(*------------------------------------------------------------------------------------------Modbus TCP Functions---------------------------------------------------------------------------------------------*)

fbMBRead_FC3(	sIPAddr:= str_IPAdress, 
				nTCPPort:= 502,
				cbLength:= SIZEOF(arrBuffer_FC3), 
				pDestAddr:= ADR(arrBuffer_FC3), 
				tTimeout:= T#10S,
				nErrId => udint_Error_ID);

FPError_FC_3(CLK:= fbMBRead_FC3.  bError, Q=> );		

(*------------------------------------------------------------------------------------------State Machine Error---------------------------------------------------------------------------------------------*)	

CASE iStateModbusError OF
	
	300://Error
		timer_Wait.IN :=TRUE;
		timer_Delay.IN := FALSE;
		fbMBRead_FC3.bExecute := FALSE;
		m_MBTCPError := TRUE; 		
		m_Poll_ok:=FALSE;
		int_Data_Received:=0;
				//Restart from new with the Read out part after an Error
		IF timer_Wait.Q = TRUE THEN
			iStateModbusRead := 0;	
			iStateModbusError := 0;
			timer_Wait.IN :=FALSE;
			timer_Timeout.IN := FALSE;
		END_IF		
							
END_CASE

END_FUNCTION_BLOCK

// ---- FBs/General/FB_ModBus_2Registers_FC4.TcPOU
FUNCTION_BLOCK FB_ModBus_2Registers_FC4
VAR_INPUT PERSISTENT
	m_Enable					: BOOL;						//Enable the Fuctionblock and his logic
	str_IPAdress				: STRING(15);				//IP Adress of the meter
	w_Adress					: WORD;						//modbus adress
	int_Divider					: INT;						//Devider of the received data
	n_UnitID					: BYTE:=255;				// dentification number of a serial sub-network device. If a device is addressed directly via TCP/IP, this value must be 16#FF / 255
	m_Float32Conversion			: BOOL;						// receives value in Float 32 / real format
	m_LittleEndian				: BOOL;

END_VAR
VAR_OUTPUT
	m_PollSuccessful			: BOOL;						//Poll succesfull		
	r_ReceivedValue				: REAL;						//Received Value
	udint_Error_ID				: UDINT;					// ERR ID FB_MBReadRegs
END_VAR
VAR
	{attribute 'hide'}
	timer_Delay					: TON;						//Timer for Delay between Requests
	{attribute 'hide'}
	timer_DelayStart			: TON;						//Timer to start the state machine with Delay after enabling or after the system ist restartet
	{attribute 'hide'}
	timer_TimeOut				: TON;						//Timer for Timeout MB Read
	{attribute 'hide'}
	iStateModbusRead			: INT;						//State machine for read out Data over Modbus RTU
	{attribute 'hide'}
	fbMBRead_FC4				: FB_MBReadInputRegs  ;		//Modbus Read Function (FC4)
	{attribute 'hide'}
	ftrig_PEnable				: f_trig;					//Internal positive Edge
	{attribute 'hide'}
	iStateModbusError			: INT;						//State machine for error out Data over Modbus TCP/IP	
	{attribute 'hide'}
	FPError_FC4				: R_TRIG;					//Internal positive Edge
	{attribute 'hide'}
	arrBuffer_FC4				: ARRAY[1..2] OF WORD;		//Buffer with Data from FC4
	{attribute 'hide'}
	timer_Connection_ok			: TON;
	int_Data_Received			: INT;
	{attribute 'hide'}
	m_MBTCPError				: BOOL;
	{attribute 'hide'}
	int_Data_Received_old		: INT;
	{attribute 'hide'}
	timer_Connection_ok_TOF	: TOF;
	{attribute 'hide'}
	fbConvertWordToDword		: FB_CV_WORD_TO_DWORD;			//Convert Word to Dword
	{attribute 'hide'}
	usintSign					: USINT;						// converstion dword to real	
	{attribute 'hide'}
	intExponent					: INT;							// converstion dword to real
	{attribute 'hide'}
	realMantisse				: REAL;							// converstion dword to real
	{attribute 'hide'}
	m_Poll_ok: BOOL;
	{attribute 'hide'}
	timer_Wait: Ton;
	int_TimeoutError: INT;
	int_FC4Error: INT;
END_VAR

(*--------------------------------------------------------------------------------------------Limits-------------------------------------------------------------------------------------*)

w_Adress := LIMIT(0,w_Adress,65535);
int_Divider := LIMIT(1,int_Divider,32767);
	
(*--------------------------------------------------------------------------------------------State Machine Read--------------------------------------------------------------------------------------*)

//Timer for Delay
timer_Delay(IN:= , PT:= T#50MS, Q=> , ET=> );

//Timeout Timer is dissabled when the Init Step is aktiv or the function is not enabled
IF iStateModbusRead = 0 OR NOT m_Enable THEN 
	timer_Timeout.IN := FALSE; 
END_IF
timer_Timeout(IN:= , PT:= T#1S, Q=> , ET=> );

//Enable with Delay that not all sockets have to be created at the same time
timer_DelayStart(IN:= m_Enable, PT:= T#1S, Q=> , ET=> );
ftrig_PEnable(CLK:= timer_DelayStart.Q, Q=> );

IF ftrig_PEnable.Q AND iStateModbusRead = 0 THEN 
	iStateModbusRead := 1; 
END_IF		
		
//Not Enabled
IF NOT m_Enable THEN 
	iStateModbusRead := 0; 
	iStateModbusError := 0; 
END_IF		
		
CASE iStateModbusRead OF

	0://Init Step 
		timer_Delay.IN := FALSE;
		fbMBRead_FC4.bExecute := FALSE;
		m_Poll_ok:=FALSE;
		int_Data_Received:=0;
	
		iStateModbusRead := 1;
	
	1://read the required registers
		//Start Read
		fbMBRead_FC4.nQuantity := 2;
		fbMBRead_FC4.nMBAddr := w_Adress;
		fbMBRead_FC4.bExecute := TRUE;
		fbMBRead_FC4.nUnitID := n_UnitID;
		timer_Timeout.IN := TRUE;
		IF fbMBRead_FC4.bBusy THEN 
			timer_Delay.IN := TRUE; 
		END_IF
		
		//Wait for Delay, copy Data and then next step
		IF NOT fbMBRead_FC4.bBusy AND NOT fbMBRead_FC4.bError AND timer_Delay.Q THEN
			m_Poll_ok:=TRUE;
			int_Data_Received:=int_Data_Received+1;
			m_MBTCPError := FALSE; 
			// convert received data
			IF m_Float32Conversion AND NOT m_LittleEndian THEN
		//		fbConvertWordToDword(wInputValue_1:= arrBuffer_FC4[1], wInputValue_2:= arrBuffer_FC4[2], eByteOrderForConvert:= eByteOrder.eLittleEndian , dwOutputValue=> );
				fbConvertWordToDword(wInputValue_1:= arrBuffer_FC4[1], wInputValue_2:= arrBuffer_FC4[2], eByteOrderForConvert:= eByteOrder.eBigEndian , dwOutputValue=> );
				(* Sign *)
				usintSign:=BOOL_TO_USINT(fbConvertWordToDword.dwOutputValue.31);
				(* Exponent *)
				intExponent:=DWORD_TO_INT(SHR(fbConvertWordToDword.dwOutputValue,23) AND 16#FF);
				(* Mantisse *)
				realMantisse:=DWORD_TO_REAL(fbConvertWordToDword.dwOutputValue AND 16#7FFFFF);
				(* Result *)
				r_ReceivedValue := LREAL_TO_REAL((EXPT((-1),usintSign) * (1+realMantisse/8388608) * EXPT(2,intExponent-127))/int_Divider);
			ELSIF m_Float32Conversion AND m_LittleEndian THEN
				fbConvertWordToDword(wInputValue_1:= arrBuffer_FC4[1], wInputValue_2:= arrBuffer_FC4[2], eByteOrderForConvert:= eByteOrder.eLittleEndian , dwOutputValue=> );
				(* Sign *)
				usintSign:=BOOL_TO_USINT(fbConvertWordToDword.dwOutputValue.31);
				(* Exponent *)
				intExponent:=DWORD_TO_INT(SHR(fbConvertWordToDword.dwOutputValue,23) AND 16#FF);
				(* Mantisse *)
				realMantisse:=DWORD_TO_REAL(fbConvertWordToDword.dwOutputValue AND 16#7FFFFF);
				(* Result *)
				r_ReceivedValue := LREAL_TO_REAL((EXPT((-1),usintSign) * (1+realMantisse/8388608) * EXPT(2,intExponent-127))/int_Divider);
			ELSE
				fbConvertWordToDword(wInputValue_1:= arrBuffer_FC4[2], wInputValue_2:= arrBuffer_FC4[1], eByteOrderForConvert:= eByteOrder.eLittleEndian , dwOutputValue=> );
				r_ReceivedValue := DINT_TO_REAL(fbConvertWordToDword.dwOutputValue)/int_Divider;
			END_IF
			
			//Go to Next Step
			timer_Timeout.IN := FALSE;
			fbMBRead_FC4.bExecute := FALSE;
			timer_Delay.IN := FALSE;		
			iStateModbusRead := 3;
		END_IF	

		//Error or Timeout
		IF FPError_FC4.Q THEN 
			iStateModbusError := 300;
			int_FC4Error := int_FC4Error+1;
		ELSIF timer_Timeout.Q THEN 
			timer_Timeout.IN := FALSE; 	  	
			iStateModbusError := 300;
			int_TimeoutError := int_TimeoutError+1;
		END_IF
		
	
	3://Wait and go to step 1
		//1 because 0 is the Init Step for Read
		timer_Wait.IN := TRUE;
		
		IF timer_Wait.Q = TRUE THEN
			iStateModbusRead := 1;
			timer_Wait.IN :=FALSE;
		END_IF

			
		
		//Error on Master, changes on Inputs or Timeout
		IF timer_Timeout.Q THEN 
			iStateModbusError := 300; 
		END_IF
	
END_CASE

(* wait timer*)

timer_Wait(PT:=T#3S);


(*------------------------------------------------------------------Error and Warning----------------------------------------------------------------------------*)	
 
timer_Connection_ok			(In:=int_Data_Received<>int_Data_Received_old,PT:=T#10S);
timer_Connection_ok_TOF		(In:=NOT(int_Data_Received<>int_Data_Received_old) AND int_Data_Received>3 ,PT:=T#20S);
int_Data_Received_old:=int_Data_Received;
m_PollSuccessful:=NOT timer_Connection_ok.Q AND timer_Connection_ok_TOF.Q ;

(*------------------------------------------------------------------------------------------Modbus TCP Functions---------------------------------------------------------------------------------------------*)

fbMBRead_FC4(	sIPAddr:= str_IPAdress, 
				nTCPPort:= 502,
				cbLength:= SIZEOF(arrBuffer_FC4), 
				pDestAddr:= ADR(arrBuffer_FC4), 
				tTimeout:= T#10S,
				nErrId => udint_Error_ID);

FPError_FC4(CLK:= fbMBRead_FC4.  bError, Q=> );		

(*------------------------------------------------------------------------------------------State Machine Error---------------------------------------------------------------------------------------------*)	

CASE iStateModbusError OF
	
	300://Error
		timer_Wait.IN :=TRUE;
		timer_Delay.IN := FALSE;
		fbMBRead_FC4.bExecute := FALSE;
		m_MBTCPError := TRUE; 		
		m_Poll_ok:=FALSE;
		int_Data_Received:=0;
				//Restart from new with the Read out part after an Error
		IF timer_Wait.Q = TRUE THEN
			iStateModbusRead := 0;	
			iStateModbusError := 0;
			timer_Wait.IN :=FALSE;
			timer_Timeout.IN := FALSE;
		END_IF		
							
END_CASE

END_FUNCTION_BLOCK

// ---- FBs/GMC Instruments/FB_EM2289.TcPOU
FUNCTION_BLOCK FB_EM2289
VAR_INPUT PERSISTENT
	m_Enable					: BOOL;						//Enable the Fuctionblock and his logic
	str_IPAdress				: STRING(15);				//IP Adress of the meter
END_VAR
VAR_OUTPUT
	real_RealPower_kW				: REAL;					// Real power in W
	real_RealPowerL1_kW				: REAL;					// Real power in W
	real_RealPowerL2_kW				: REAL;					// Real power in W
	real_RealPowerL3_kW				: REAL;					// Real power in W
	real_ReactivePower_kVAr			: REAL;					// Reactive power in VAr
	real_ApparentPower_kVA			: REAL;					// Apparent power in VA
	real_Frequency_Hz				: REAL;					// Frequency in Hz
	real_VoltageL1N_V				: REAL;					//  Voltage L1-N in V 
	real_VoltageL2N_V				: REAL;					//  Voltage L2-N in V 
	real_VoltageL3N_V				: REAL;					//  Voltage L3-N in V 
	real_VoltageL1L2_V				: REAL;					//  Voltage L1-L2 in V 
	real_VoltageL2L3_V				: REAL;					//  Voltage L2-L3 in V 
	real_VoltageL3L1_V				: REAL;					//  Voltage L3-L1 in V 
	real_CurrentL1_A				: REAL;					//  Current L1 in A
	real_CurrentL2_A				: REAL;					//  Current L2 in A
	real_CurrentL3_A				: REAL;					//  Current L3 in A
	real_EnergyTotal_Import_Wh		: REAL;					// Energy total in Wh
	real_EnergyTotal_Export_Wh		: REAL;					// Energy total in Wh
	real_EnergyTotal_ExportT1_Wh	: REAL;					// Energy total in Wh
	real_EnergyTotal_ExportT2_Wh	: REAL;					// Energy total in Wh
	m_PollSuccessful				: BOOL;					// Poll succesfull		
	udint_Error_ID					: UDINT;				// ERR ID FB_MBReadRegs
END_VAR
VAR
	{attribute 'hide'}
	w_Adress					: WORD;						//modbus adress
	{attribute 'hide'}
	usint_Quantity				: USINT;					//Number of Words to get polled, max 100
	{attribute 'hide'}
	fbConvertWordToDword		: FB_CV_WORD_TO_DWORD;			//Convert Word to Dword
	{attribute 'hide'}
	usintSign					: USINT;						// converstion dword to real	
	{attribute 'hide'}
	intExponent					: INT;							// converstion dword to real
	{attribute 'hide'}
	realMantisse				: REAL;							// converstion dword to real
	{attribute 'hide'}
	timer_Delay					: TON;						//Timer for Delay between Requests
	{attribute 'hide'}
	timer_DelayStart			: TON;						//Timer to start the state machine with Delay after enabling or after the system ist restartet
	{attribute 'hide'}
	timer_TimeOut				: TON;						//Timer for Timeout MB Read
	{attribute 'hide'}
	iStateModbusRead			: INT;						//State machine for read out Data over Modbus RTU
	{attribute 'hide'}
	fbMBRead_FC4				: FB_MBReadInputRegs  ;		//Modbus Read Function (FC4)
	{attribute 'hide'}
	ftrig_PEnable				: f_trig;					//Internal positive Edge
	{attribute 'hide'}
	iStateModbusError			: INT;						//State machine for error out Data over Modbus TCP/IP	
	{attribute 'hide'}
	FPError_FC_4				: R_TRIG;					//Internal positive Edge
	{attribute 'hide'}
	arrBuffer_FC4				: ARRAY[0..100] OF WORD;		//Buffer with Data from FC4
	{attribute 'hide'}
	timer_Connection_ok			: TON;
	{attribute 'hide'}
	int_Data_Received			: INT;
	{attribute 'hide'}
	m_MBTCPError				: BOOL;
	{attribute 'hide'}
	int_Data_Received_old		: INT;
	{attribute 'hide'}
	timer_Connection_ok_TOF	: TOF;
	{attribute 'hide'}
	m_Poll_ok: BOOL;
	{attribute 'hide'}
	timer_Wait: Ton;
	{attribute 'hide'}
	int_TimeoutError: INT;
	{attribute 'hide'}
	int_FC4Error: INT;
	{attribute 'hide'}
	i: INT;
	{attribute 'hide'}
	x: INT;
	sint_Exponent: SINT;
	real_EnergyFactor: REAL;
	
END_VAR

// v0.1 by Stefan Lackner 20230327
// not tested 
// reads out GMC Instruments EM2289   


(*--------------------------------------------------------------------------------------------Limits-------------------------------------------------------------------------------------*)
w_Adress := LIMIT(0,w_Adress,65000);
usint_Quantity := LIMIT(1,usint_Quantity,100);
	
(*--------------------------------------------------------------------------------------------State Machine Read--------------------------------------------------------------------------------------*)

//Timer for Delay
timer_Delay(IN:= , PT:= T#50MS, Q=> , ET=> );

//Timeout Timer is dissabled when the Init Step is aktiv or the function is not enabled
IF iStateModbusRead = 0 OR NOT m_Enable THEN 
	timer_Timeout.IN := FALSE; 
END_IF
timer_Timeout(IN:= , PT:= T#1S, Q=> , ET=> );

//Enable with Delay that not all sockets have to be created at the same time
timer_DelayStart(IN:= m_Enable, PT:= T#1S, Q=> , ET=> );
ftrig_PEnable(CLK:= timer_DelayStart.Q, Q=> );

IF ftrig_PEnable.Q AND iStateModbusRead = 0 THEN 
	iStateModbusRead := 1; 
END_IF		
		
//Not Enabled
IF NOT m_Enable THEN 
	iStateModbusRead := 0; 
	iStateModbusError := 0; 
END_IF		
		
CASE iStateModbusRead OF

	0://Init Step 
		timer_Delay.IN := FALSE;
		fbMBRead_FC4.bExecute := FALSE;
		m_Poll_ok:=FALSE;
		int_Data_Received:=0;
		iStateModbusRead := iStateModbusRead+1;

	1: // clean the array  Poll 1
		FOR i:=0 TO 100 BY 1 DO
			arrBuffer_FC4[i] := 0;
		END_FOR
		w_Adress := 0;
		usint_Quantity := 13; 
		iStateModbusRead := iStateModbusRead+1;
		
	2://read the required registers
		//Start Read Poll 1
		fbMBRead_FC4.nQuantity := usint_Quantity;
		fbMBRead_FC4.nMBAddr := w_Adress;
		fbMBRead_FC4.bExecute := TRUE;
		fbMBRead_FC4.nUnitID := 1;
		timer_Timeout.IN := TRUE;
		IF fbMBRead_FC4.bBusy THEN 
			timer_Delay.IN := TRUE; 
		END_IF
		
		//Wait for Delay, copy Data and then next step
		IF NOT fbMBRead_FC4.bBusy AND NOT fbMBRead_FC4.bError AND timer_Delay.Q THEN
			m_Poll_ok:=TRUE;
			int_Data_Received:=int_Data_Received+1;
			m_MBTCPError := FALSE; 
			
			//Go to Next Step
			timer_Timeout.IN := FALSE;
			fbMBRead_FC4.bExecute := FALSE;
			timer_Delay.IN := FALSE;		
			iStateModbusRead := iStateModbusRead+1;
		END_IF	

		//Error or Timeout
		IF FPError_FC_4.Q THEN 
			iStateModbusError := 300;
			int_FC4Error := int_FC4Error+1;
		ELSIF timer_Timeout.Q THEN  
			timer_Timeout.IN := FALSE; 	
			iStateModbusError := 300;
			int_TimeoutError := int_TimeoutError+1;
		END_IF
		
	3: // convert data Poll 1
		sint_Exponent := WORD_TO_SINT (arrBuffer_FC4[12]);
		real_VoltageL1L2_V := LREAL_TO_REAL(WORD_TO_REAL(arrBuffer_FC4[0])* EXPT (10,sint_Exponent));
		real_VoltageL2L3_V := LREAL_TO_REAL(WORD_TO_REAL(arrBuffer_FC4[1])* EXPT (10,sint_Exponent));
		real_VoltageL3L1_V := LREAL_TO_REAL(WORD_TO_REAL(arrBuffer_FC4[2])* EXPT (10,sint_Exponent));
		real_VoltageL1N_V :=  LREAL_TO_REAL(WORD_TO_REAL(arrBuffer_FC4[4])* EXPT (10,sint_Exponent));
		real_VoltageL2N_V :=  LREAL_TO_REAL(WORD_TO_REAL(arrBuffer_FC4[5])* EXPT (10,sint_Exponent));
		real_VoltageL3N_V :=  LREAL_TO_REAL(WORD_TO_REAL(arrBuffer_FC4[6])* EXPT (10,sint_Exponent));
		real_Frequency_Hz := WORD_TO_REAL(arrBuffer_FC4[11])/100;
		// go to next step
		iStateModbusRead := iStateModbusRead+1;
	
	4://Wait and go to next step
		timer_Wait.IN := TRUE;
		
		IF timer_Wait.Q = TRUE THEN
			iStateModbusRead := iStateModbusRead+1;
			timer_Wait.IN :=FALSE;
		END_IF

	5: // clean the array  Poll 2
		FOR i:=0 TO 100 BY 1 DO
			arrBuffer_FC4[i] := 0;
		END_FOR
		w_Adress := 100;
		usint_Quantity := 9; 
		iStateModbusRead := iStateModbusRead+1;
		
	6://read the required registers
		//Start Read  Poll 2
		fbMBRead_FC4.nQuantity := usint_Quantity;
		fbMBRead_FC4.nMBAddr := w_Adress;
		fbMBRead_FC4.bExecute := TRUE;
		fbMBRead_FC4.nUnitID := 1;
		timer_Timeout.IN := TRUE;
		IF fbMBRead_FC4.bBusy THEN 
			timer_Delay.IN := TRUE; 
		END_IF
		
		//Wait for Delay, copy Data and then next step
		IF NOT fbMBRead_FC4.bBusy AND NOT fbMBRead_FC4.bError AND timer_Delay.Q THEN
			m_Poll_ok:=TRUE;
			int_Data_Received:=int_Data_Received+1;
			m_MBTCPError := FALSE; 
			
			//Go to Next Step
			timer_Timeout.IN := FALSE;
			fbMBRead_FC4.bExecute := FALSE;
			timer_Delay.IN := FALSE;		
			iStateModbusRead := iStateModbusRead+1;
		END_IF	

		//Error or Timeout
		IF FPError_FC_4.Q THEN 
			iStateModbusError := 300;
			int_FC4Error := int_FC4Error+1;
		ELSIF timer_Timeout.Q THEN  
			timer_Timeout.IN := FALSE; 	
			iStateModbusError := 300;
			int_TimeoutError := int_TimeoutError+1;
		END_IF
		
	7: // convert data Poll 2
		sint_Exponent := WORD_TO_SINT (arrBuffer_FC4[8]);
		real_CurrentL1_A := LREAL_TO_REAL(WORD_TO_REAL(arrBuffer_FC4[0])* EXPT (10,sint_Exponent));
		real_CurrentL2_A := LREAL_TO_REAL(WORD_TO_REAL(arrBuffer_FC4[1])* EXPT (10,sint_Exponent));
		real_CurrentL3_A := LREAL_TO_REAL(WORD_TO_REAL(arrBuffer_FC4[2])* EXPT (10,sint_Exponent));
		
		// go to next step
		iStateModbusRead := iStateModbusRead+1;
			
		//Error on Master, changes on Inputs or Timeout
		IF timer_Timeout.Q THEN 
			iStateModbusError := 300; 
		END_IF
		
	8://Wait and go to next step
		timer_Wait.IN := TRUE;
		
		IF timer_Wait.Q = TRUE THEN
			iStateModbusRead := iStateModbusRead+1;
			timer_Wait.IN :=FALSE;
		END_IF

	9: // clean the array  Poll 3
		FOR i:=0 TO 100 BY 1 DO
			arrBuffer_FC4[i] := 0;
		END_FOR
		w_Adress := 200;
		usint_Quantity := 13; 
		iStateModbusRead := iStateModbusRead+1;
		
	10://read the required registers
		//Start Read  Poll 3
		fbMBRead_FC4.nQuantity := usint_Quantity;
		fbMBRead_FC4.nMBAddr := w_Adress;
		fbMBRead_FC4.bExecute := TRUE;
		fbMBRead_FC4.nUnitID := 1;
		timer_Timeout.IN := TRUE;
		IF fbMBRead_FC4.bBusy THEN 
			timer_Delay.IN := TRUE; 
		END_IF
		
		//Wait for Delay, copy Data and then next step
		IF NOT fbMBRead_FC4.bBusy AND NOT fbMBRead_FC4.bError AND timer_Delay.Q THEN
			m_Poll_ok:=TRUE;
			int_Data_Received:=int_Data_Received+1;
			m_MBTCPError := FALSE; 
			
			//Go to Next Step
			timer_Timeout.IN := FALSE;
			fbMBRead_FC4.bExecute := FALSE;
			timer_Delay.IN := FALSE;		
			iStateModbusRead := iStateModbusRead+1;
		END_IF	

		//Error or Timeout
		IF FPError_FC_4.Q THEN 
			iStateModbusError := 300;
			int_FC4Error := int_FC4Error+1;
		ELSIF timer_Timeout.Q THEN  
			timer_Timeout.IN := FALSE; 	
			iStateModbusError := 300;
			int_TimeoutError := int_TimeoutError+1;
		END_IF
		
	11: // convert data Poll 3
		sint_Exponent := WORD_TO_SINT (arrBuffer_FC4[12]);
		real_RealPowerL1_kW := LREAL_TO_REAL(WORD_TO_REAL(arrBuffer_FC4[0])* EXPT (10,sint_Exponent)/1000);
		real_RealPowerL2_kW := LREAL_TO_REAL(WORD_TO_REAL(arrBuffer_FC4[1])* EXPT (10,sint_Exponent)/1000);
		real_RealPowerL3_kW := LREAL_TO_REAL(WORD_TO_REAL(arrBuffer_FC4[2])* EXPT (10,sint_Exponent)/1000);
		real_RealPower_kW := LREAL_TO_REAL(WORD_TO_REAL(arrBuffer_FC4[3])* EXPT (10,sint_Exponent)/1000);
		real_RealPowerL1_kW := LREAL_TO_REAL(WORD_TO_REAL(arrBuffer_FC4[0])* EXPT (10,sint_Exponent)/1000);
		real_ReactivePower_kVAr := LREAL_TO_REAL(WORD_TO_REAL(arrBuffer_FC4[7])* EXPT (10,sint_Exponent)/1000);
		
		IF (real_RealPower_kW*real_RealPower_kW + real_ReactivePower_kVAr*real_ReactivePower_kVAr) <>0 THEN 
			real_ApparentPower_kVA := SQRT(ABS(real_RealPower_kW*real_RealPower_kW + real_ReactivePower_kVAr*real_ReactivePower_kVAr));	
		ELSE
	 		real_ApparentPower_kVA :=0;
		END_IF
		
		
		// go to next step
		iStateModbusRead := iStateModbusRead+1;
			
		//Error on Master, changes on Inputs or Timeout
		IF timer_Timeout.Q THEN 
			iStateModbusError := 300; 
		END_IF
		
	12://Wait and go to next step
		timer_Wait.IN := TRUE;
		
		IF timer_Wait.Q = TRUE THEN
			iStateModbusRead := iStateModbusRead+1;
			timer_Wait.IN :=FALSE;
		END_IF

	13: // clean the array  Poll 4
		FOR i:=0 TO 100 BY 1 DO
			arrBuffer_FC4[i] := 0;
		END_FOR
		w_Adress := 300;
		usint_Quantity := 10; 
		iStateModbusRead := iStateModbusRead+1;
		
	14://read the required registers
		//Start Read  Poll 4
		fbMBRead_FC4.nQuantity := usint_Quantity;
		fbMBRead_FC4.nMBAddr := w_Adress;
		fbMBRead_FC4.bExecute := TRUE;
		fbMBRead_FC4.nUnitID := 1;
		timer_Timeout.IN := TRUE;
		IF fbMBRead_FC4.bBusy THEN 
			timer_Delay.IN := TRUE; 
		END_IF
		
		//Wait for Delay, copy Data and then next step
		IF NOT fbMBRead_FC4.bBusy AND NOT fbMBRead_FC4.bError AND timer_Delay.Q THEN
			m_Poll_ok:=TRUE;
			int_Data_Received:=int_Data_Received+1;
			m_MBTCPError := FALSE; 
			
			//Go to Next Step
			timer_Timeout.IN := FALSE;
			fbMBRead_FC4.bExecute := FALSE;
			timer_Delay.IN := FALSE;		
			iStateModbusRead := iStateModbusRead+1;
		END_IF	

		//Error or Timeout
		IF FPError_FC_4.Q THEN 
			iStateModbusError := 300;
			int_FC4Error := int_FC4Error+1;
		ELSIF timer_Timeout.Q THEN  
			timer_Timeout.IN := FALSE; 	
			iStateModbusError := 300;
			int_TimeoutError := int_TimeoutError+1;
		END_IF
		
	15: // convert data Poll 4
		// energy factor
		fbConvertWordToDword(wInputValue_1:= arrBuffer_FC4[8], wInputValue_2:= arrBuffer_FC4[9], eByteOrderForConvert:= eByteOrder.eBigEndian , dwOutputValue=> );
		real_EnergyFactor := DWORD_TO_REAL (fbConvertWordToDword.dwOutputValue);
				
		fbConvertWordToDword(wInputValue_1:= arrBuffer_FC4[0], wInputValue_2:= arrBuffer_FC4[1], eByteOrderForConvert:= eByteOrder.eBigEndian , dwOutputValue=> );
		real_EnergyTotal_Import_Wh := DWORD_TO_REAL(fbConvertWordToDword.dwOutputValue) * real_EnergyFactor;
		
		fbConvertWordToDword(wInputValue_1:= arrBuffer_FC4[2], wInputValue_2:= arrBuffer_FC4[3], eByteOrderForConvert:= eByteOrder.eBigEndian , dwOutputValue=> );
		real_EnergyTotal_Export_Wh := DWORD_TO_REAL(fbConvertWordToDword.dwOutputValue) * real_EnergyFactor;
	
		// go to next step
		iStateModbusRead := iStateModbusRead+1;
			
		//Error on Master, changes on Inputs or Timeout
		IF timer_Timeout.Q THEN 
			iStateModbusError := 300; 
		END_IF		

	16://Wait and go to next step
		timer_Wait.IN := TRUE;
		
		IF timer_Wait.Q = TRUE THEN
			iStateModbusRead := iStateModbusRead+1;
			timer_Wait.IN :=FALSE;
		END_IF

	17: // clean the array  Poll 5
		FOR i:=0 TO 100 BY 1 DO
			arrBuffer_FC4[i] := 0;
		END_FOR
		w_Adress := 600;
		usint_Quantity := 10; 
		iStateModbusRead := iStateModbusRead+1;
		
	18://read the required registers
		//Start Read  Poll 5
		fbMBRead_FC4.nQuantity := usint_Quantity;
		fbMBRead_FC4.nMBAddr := w_Adress;
		fbMBRead_FC4.bExecute := TRUE;
		fbMBRead_FC4.nUnitID := 1;
		timer_Timeout.IN := TRUE;
		IF fbMBRead_FC4.bBusy THEN 
			timer_Delay.IN := TRUE; 
		END_IF
		
		//Wait for Delay, copy Data and then next step
		IF NOT fbMBRead_FC4.bBusy AND NOT fbMBRead_FC4.bError AND timer_Delay.Q THEN
			m_Poll_ok:=TRUE;
			int_Data_Received:=int_Data_Received+1;
			m_MBTCPError := FALSE; 
			
			//Go to Next Step
			timer_Timeout.IN := FALSE;
			fbMBRead_FC4.bExecute := FALSE;
			timer_Delay.IN := FALSE;		
			iStateModbusRead := iStateModbusRead+1;
		END_IF	

		//Error or Timeout
		IF FPError_FC_4.Q THEN 
			iStateModbusError := 300;
			int_FC4Error := int_FC4Error+1;
		ELSIF timer_Timeout.Q THEN  
			timer_Timeout.IN := FALSE; 	
			iStateModbusError := 300;
			int_TimeoutError := int_TimeoutError+1;
		END_IF
		
	19: // convert data Poll 5
		// energy factor
		fbConvertWordToDword(wInputValue_1:= arrBuffer_FC4[8], wInputValue_2:= arrBuffer_FC4[9], eByteOrderForConvert:= eByteOrder.eBigEndian , dwOutputValue=> );
		real_EnergyFactor := DWORD_TO_REAL (fbConvertWordToDword.dwOutputValue);
				
		fbConvertWordToDword(wInputValue_1:= arrBuffer_FC4[2], wInputValue_2:= arrBuffer_FC4[3], eByteOrderForConvert:= eByteOrder.eBigEndian , dwOutputValue=> );
		real_EnergyTotal_ExportT1_Wh := DWORD_TO_REAL(fbConvertWordToDword.dwOutputValue) * real_EnergyFactor;
		
		fbConvertWordToDword(wInputValue_1:= arrBuffer_FC4[6], wInputValue_2:= arrBuffer_FC4[7], eByteOrderForConvert:= eByteOrder.eBigEndian , dwOutputValue=> );
		real_EnergyTotal_ExportT2_Wh := DWORD_TO_REAL(fbConvertWordToDword.dwOutputValue) * real_EnergyFactor;
				
		// go to next step
		iStateModbusRead := iStateModbusRead+1;
			
		//Error on Master, changes on Inputs or Timeout
		IF timer_Timeout.Q THEN 
			iStateModbusError := 300; 
		END_IF		

	20://Wait and go to next step
		timer_Wait.IN := TRUE;
		
		IF timer_Wait.Q = TRUE THEN
			iStateModbusRead := 1;
			timer_Wait.IN :=FALSE;
		END_IF
	
END_CASE

(* wait timer*)

timer_Wait(PT:=T#1S);


(*------------------------------------------------------------------Error and Warning----------------------------------------------------------------------------*)	
 
timer_Connection_ok			(In:=int_Data_Received<>int_Data_Received_old,PT:=T#10S);
timer_Connection_ok_TOF		(In:=NOT(int_Data_Received<>int_Data_Received_old) AND int_Data_Received>3 ,PT:=T#20S);
int_Data_Received_old:=int_Data_Received;
m_PollSuccessful:=NOT timer_Connection_ok.Q AND timer_Connection_ok_TOF.Q ;

(*------------------------------------------------------------------------------------------Modbus TCP Functions---------------------------------------------------------------------------------------------*)

fbMBRead_FC4(	sIPAddr:= str_IPAdress, 
				nTCPPort:= 502,
				cbLength:= SIZEOF(arrBuffer_FC4), 
				pDestAddr:= ADR(arrBuffer_FC4), 
				tTimeout:= T#10S,
				nErrId => udint_Error_ID);

FPError_FC_4(CLK:= fbMBRead_FC4.bError, Q=> );		

(*------------------------------------------------------------------------------------------State Machine Error---------------------------------------------------------------------------------------------*)	

CASE iStateModbusError OF
	
	300://Error
		timer_Wait.IN :=TRUE;
		timer_Delay.IN := FALSE;
		fbMBRead_FC4.bExecute := FALSE;
		m_MBTCPError := TRUE; 		
		m_Poll_ok:=FALSE;
		int_Data_Received:=0;
				//Restart from new with the Read out part after an Error
		IF timer_Wait.Q = TRUE THEN
			iStateModbusRead := 0;	
			iStateModbusError := 0;
			timer_Wait.IN :=FALSE;
			timer_Timeout.IN := FALSE;
		END_IF		
							
END_CASE

END_FUNCTION_BLOCK

// ---- FBs/GossenMetrawatt/FB_ENERGYMID_EM22xx_23xx.TcPOU
FUNCTION_BLOCK FB_ENERGYMID_EM22xx_23xx
VAR_INPUT PERSISTENT
	m_Enable					: BOOL;						//Enable the Fuctionblock and his logic
	str_IPAdress				: STRING(15);				//IP Adress of the meter
END_VAR
VAR_OUTPUT
	real_RealPower_kW				: REAL;					// Real power in W
	real_RealPowerL1_kW				: REAL;					// Real power in W
	real_RealPowerL2_kW				: REAL;					// Real power in W
	real_RealPowerL3_kW				: REAL;					// Real power in W
	real_ReactivePowerL1_kVAr		: REAL;					// Reactive power in kVAr
	real_ReactivePowerL2_kVAr		: REAL;					// Reactive power in kVAr
	real_ReactivePowerL3_kVAr		: REAL;					// Reactive power in kVAr	
	real_ReactivePower_kVAr			: REAL;					// Reactive power in kVAr
	real_PowerFactorL1				: REAL;					// Power Factor
	real_PowerFactorL2				: REAL;					// Power Factor
	real_PowerFactorL3				: REAL;					// Power Factor	
	real_PowerFactor				: REAL;					// Power Factor
	real_Frequency_Hz				: REAL;					// Frequency in Hz
	real_VoltageL1N_V				: REAL;					//  Voltage L1-N in V 
	real_VoltageL2N_V				: REAL;					//  Voltage L2-N in V 
	real_VoltageL3N_V				: REAL;					//  Voltage L3-N in V 
	real_VoltageL1L2_V				: REAL;					//  Voltage L1-L2 in V 
	real_VoltageL2L3_V				: REAL;					//  Voltage L2-L3 in V 
	real_VoltageL3L1_V				: REAL;					//  Voltage L3-L1 in V 
	real_CurrentL1_A				: REAL;					//  Current L1 in A
	real_CurrentL2_A				: REAL;					//  Current L2 in A
	real_CurrentL3_A				: REAL;					//  Current L3 in A
	real_EnergyTotal_Import_kWh		: REAL;					// Energy total in Wh
	real_EnergyTotal_Export_kWh		: REAL;					// Energy total in Wh
	
	m_PollSuccessful				: BOOL;					// Poll succesfull		
	udint_Error_ID					: UDINT;				// ERR ID FB_MBReadRegs
END_VAR
VAR
	{attribute 'hide'}
	w_Adress					: WORD;						//modbus adress
	{attribute 'hide'}
	usint_Quantity				: USINT;					//Number of Words to get polled, max 100
	{attribute 'hide'}
	fbConvertWordToDword		: FB_CV_WORD_TO_DWORD;			//Convert Word to Dword
	{attribute 'hide'}
	usintSign					: USINT;						// converstion dword to real	
	{attribute 'hide'}
	intExponent					: INT;							// converstion dword to real
	{attribute 'hide'}
	realMantisse				: REAL;							// converstion dword to real
	{attribute 'hide'}
	timer_Delay					: TON;						//Timer for Delay between Requests
	{attribute 'hide'}
	timer_DelayStart			: TON;						//Timer to start the state machine with Delay after enabling or after the system ist restartet
	{attribute 'hide'}
	timer_TimeOut				: TON;						//Timer for Timeout MB Read
	{attribute 'hide'}
	iStateModbusRead			: INT;						//State machine for read out Data over Modbus RTU
	{attribute 'hide'}
	fbMBRead_FC4				: FB_MBReadInputRegs;		//Modbus Read Function (FC4)
	{attribute 'hide'}
	ftrig_PEnable				: f_trig;					//Internal positive Edge
	{attribute 'hide'}
	iStateModbusError			: INT;						//State machine for error out Data over Modbus TCP/IP	
	{attribute 'hide'}
	FPError_FC_4				: R_TRIG;					//Internal positive Edge
	{attribute 'hide'}
	arrBuffer_FC4				: ARRAY[0..11] OF WORD;		//Buffer with Data from FC4
	{attribute 'hide'}
	arrBuffer_Received			: ARRAY[0..310] OF WORD;		//Total received Data
	{attribute 'hide'}
	timer_Connection_ok			: TON;
	{attribute 'hide'}
	int_Data_Received			: INT;
	{attribute 'hide'}
	m_MBTCPError				: BOOL;
	{attribute 'hide'}
	int_Data_Received_old		: INT;
	{attribute 'hide'}
	timer_Connection_ok_TOF	: TOF;
	{attribute 'hide'}
	m_Poll_ok: BOOL;
	{attribute 'hide'}
	timer_Wait: Ton;
	{attribute 'hide'}
	int_TimeoutError: INT;
	{attribute 'hide'}
	int_FC4Error: INT;
	{attribute 'hide'}
	i: INT;
END_VAR

// v0.1 by Markus Schwarzmann 20240627
// reads out Gossen Metrawatt ENERGYMID EM2281/EM2289/EM2381/EM2387/EM2389


(*--------------------------------------------------------------------------------------------Limits-------------------------------------------------------------------------------------*)
w_Adress := LIMIT(0,w_Adress,65000);
usint_Quantity := LIMIT(1,usint_Quantity,100);
	
(*--------------------------------------------------------------------------------------------State Machine Read--------------------------------------------------------------------------------------*)

//Timer for Delay
timer_Delay(IN:= , PT:= T#50MS, Q=> , ET=> );

//Timeout Timer is dissabled when the Init Step is aktiv or the function is not enabled
IF iStateModbusRead = 0 OR NOT m_Enable THEN 
	timer_Timeout.IN := FALSE; 
END_IF
timer_Timeout(IN:= , PT:= T#1S, Q=> , ET=> );

//Enable with Delay that not all sockets have to be created at the same time
timer_DelayStart(IN:= m_Enable, PT:= T#1S, Q=> , ET=> );
ftrig_PEnable(CLK:= timer_DelayStart.Q, Q=> );

IF ftrig_PEnable.Q AND iStateModbusRead = 0 THEN 
	iStateModbusRead := 1; 
END_IF		
		
//Not Enabled
IF NOT m_Enable THEN 
	iStateModbusRead := 0; 
	iStateModbusError := 0; 
END_IF		
		
CASE iStateModbusRead OF

	0://Init Step 
		timer_Delay.IN := FALSE;
		fbMBRead_FC4.bExecute := FALSE;
		m_Poll_ok:=FALSE;
		int_Data_Received:=0;
		iStateModbusRead := iStateModbusRead+1;

	1: // clean the array  Poll 1
		FOR i:=0 TO 11 BY 1 DO
			arrBuffer_FC4[i] := 0;
		END_FOR
		w_Adress := 0;
		usint_Quantity := 12; 
		iStateModbusRead := iStateModbusRead+1;
		
	2://read the required registers
		//Start Read Poll 1, Voltage
		fbMBRead_FC4.nQuantity := usint_Quantity;
		fbMBRead_FC4.nMBAddr := w_Adress;
		fbMBRead_FC4.bExecute := TRUE;
		fbMBRead_FC4.nUnitID := 1;
		timer_Timeout.IN := TRUE;
		IF fbMBRead_FC4.bBusy THEN 
			timer_Delay.IN := TRUE; 
		END_IF
		
		//Wait for Delay, copy Data and then next step
		IF NOT fbMBRead_FC4.bBusy AND NOT fbMBRead_FC4.bError AND timer_Delay.Q THEN
			m_Poll_ok:=TRUE;
			int_Data_Received:=int_Data_Received+1;
			m_MBTCPError := FALSE; 
			
			FOR i:=0 TO 11 BY 1 DO
				arrBuffer_Received[i + WORD_TO_INT(w_Adress)] := arrBuffer_FC4[i];
			END_FOR
			
			//Go to Next Step
			timer_Timeout.IN := FALSE;
			fbMBRead_FC4.bExecute := FALSE;
			timer_Delay.IN := FALSE;		
			iStateModbusRead := iStateModbusRead+1;
		END_IF	

		//Error or Timeout
		IF FPError_FC_4.Q THEN 
			iStateModbusError := 300;
			int_FC4Error := int_FC4Error+1;
		ELSIF timer_Timeout.Q THEN  
			timer_Timeout.IN := FALSE; 	
			iStateModbusError := 300;
			int_TimeoutError := int_TimeoutError+1;
		END_IF
	
	3://Wait and go to next step
		timer_Wait.IN := TRUE;
		
		IF timer_Wait.Q = TRUE THEN
			iStateModbusRead := iStateModbusRead+1;
			timer_Wait.IN :=FALSE;
		END_IF

	4: // clean the array  Poll 2
		FOR i:=0 TO 11 BY 1 DO
			arrBuffer_FC4[i] := 0;
		END_FOR
		w_Adress := w_Adress + 100;
		usint_Quantity := 3; 
		iStateModbusRead := iStateModbusRead+1;
		
	5://read the required registers
		//Start Read Poll 2, Current
		fbMBRead_FC4.nQuantity := usint_Quantity;
		fbMBRead_FC4.nMBAddr := w_Adress;
		fbMBRead_FC4.bExecute := TRUE;
		fbMBRead_FC4.nUnitID := 1;
		timer_Timeout.IN := TRUE;
		IF fbMBRead_FC4.bBusy THEN 
			timer_Delay.IN := TRUE; 
		END_IF
		
		//Wait for Delay, copy Data and then next step
		IF NOT fbMBRead_FC4.bBusy AND NOT fbMBRead_FC4.bError AND timer_Delay.Q THEN
			m_Poll_ok:=TRUE;
			int_Data_Received:=int_Data_Received+1;
			m_MBTCPError := FALSE; 
			
			FOR i:=0 TO 11 BY 1 DO
				arrBuffer_Received[i + WORD_TO_INT(w_Adress)] := arrBuffer_FC4[i];
			END_FOR
			
			//Go to Next Step
			timer_Timeout.IN := FALSE;
			fbMBRead_FC4.bExecute := FALSE;
			timer_Delay.IN := FALSE;		
			iStateModbusRead := iStateModbusRead+1;
		END_IF	

		//Error or Timeout
		IF FPError_FC_4.Q THEN 
			iStateModbusError := 300;
			int_FC4Error := int_FC4Error+1;
		ELSIF timer_Timeout.Q THEN  
			timer_Timeout.IN := FALSE; 	
			iStateModbusError := 300;
			int_TimeoutError := int_TimeoutError+1;
		END_IF
	
	6://Wait and go to next step
		timer_Wait.IN := TRUE;
		
		IF timer_Wait.Q = TRUE THEN
			iStateModbusRead := iStateModbusRead+1;
			timer_Wait.IN :=FALSE;
		END_IF
		
	7: // clean the array  Poll 3
		FOR i:=0 TO 11 BY 1 DO
			arrBuffer_FC4[i] := 0;
		END_FOR
		w_Adress := w_Adress + 100;
		usint_Quantity := 12; 
		iStateModbusRead := iStateModbusRead+1;
		
	8://read the required registers
		//Start Read Poll 3, Power
		fbMBRead_FC4.nQuantity := usint_Quantity;
		fbMBRead_FC4.nMBAddr := w_Adress;
		fbMBRead_FC4.bExecute := TRUE;
		fbMBRead_FC4.nUnitID := 1;
		timer_Timeout.IN := TRUE;
		IF fbMBRead_FC4.bBusy THEN 
			timer_Delay.IN := TRUE; 
		END_IF
		
		//Wait for Delay, copy Data and then next step
		IF NOT fbMBRead_FC4.bBusy AND NOT fbMBRead_FC4.bError AND timer_Delay.Q THEN
			m_Poll_ok:=TRUE;
			int_Data_Received:=int_Data_Received+1;
			m_MBTCPError := FALSE; 
			
			FOR i:=0 TO 11 BY 1 DO
				arrBuffer_Received[i + WORD_TO_INT(w_Adress)] := arrBuffer_FC4[i];
			END_FOR
			
			//Go to Next Step
			timer_Timeout.IN := FALSE;
			fbMBRead_FC4.bExecute := FALSE;
			timer_Delay.IN := FALSE;		
			iStateModbusRead := iStateModbusRead+1;
		END_IF	

		//Error or Timeout
		IF FPError_FC_4.Q THEN 
			iStateModbusError := 300;
			int_FC4Error := int_FC4Error+1;
		ELSIF timer_Timeout.Q THEN  
			timer_Timeout.IN := FALSE; 	
			iStateModbusError := 300;
			int_TimeoutError := int_TimeoutError+1;
		END_IF
	
	9://Wait and go to next step
		timer_Wait.IN := TRUE;
		
		IF timer_Wait.Q = TRUE THEN
			iStateModbusRead := iStateModbusRead+1;
			timer_Wait.IN :=FALSE;
		END_IF
		
	10: // clean the array  Poll 4
		FOR i:=0 TO 11 BY 1 DO
			arrBuffer_FC4[i] := 0;
		END_FOR
		w_Adress := w_Adress + 100;
		usint_Quantity := 4; 
		iStateModbusRead := iStateModbusRead+1;
		
	11://read the required registers
		//Start Read Poll 4, Total Energy
		fbMBRead_FC4.nQuantity := usint_Quantity;
		fbMBRead_FC4.nMBAddr := w_Adress;
		fbMBRead_FC4.bExecute := TRUE;
		fbMBRead_FC4.nUnitID := 1;
		timer_Timeout.IN := TRUE;
		IF fbMBRead_FC4.bBusy THEN 
			timer_Delay.IN := TRUE; 
		END_IF
		
		//Wait for Delay, copy Data and then next step
		IF NOT fbMBRead_FC4.bBusy AND NOT fbMBRead_FC4.bError AND timer_Delay.Q THEN
			m_Poll_ok:=TRUE;
			int_Data_Received:=int_Data_Received+1;
			m_MBTCPError := FALSE; 
			
			FOR i:=0 TO 11 BY 1 DO
				arrBuffer_Received[i + WORD_TO_INT(w_Adress)] := arrBuffer_FC4[i];
			END_FOR
			
			//Go to Next Step
			timer_Timeout.IN := FALSE;
			fbMBRead_FC4.bExecute := FALSE;
			timer_Delay.IN := FALSE;		
			iStateModbusRead := 30;
		END_IF	

		//Error or Timeout
		IF FPError_FC_4.Q THEN 
			iStateModbusError := 300;
			int_FC4Error := int_FC4Error+1;
		ELSIF timer_Timeout.Q THEN  
			timer_Timeout.IN := FALSE; 	
			iStateModbusError := 300;
			int_TimeoutError := int_TimeoutError+1;
		END_IF
(*	
	12://Wait and go to next step
		timer_Wait.IN := TRUE;
		
		IF timer_Wait.Q = TRUE THEN
			iStateModbusRead := iStateModbusRead+1;
			timer_Wait.IN :=FALSE;
		END_IF		
		
	13: // clean the array  Poll 4
		FOR i:=0 TO 11 BY 1 DO
			arrBuffer_FC4[i] := 0;
		END_FOR
		w_Adress := w_Adress + 10;
		usint_Quantity := 10; 
		iStateModbusRead := iStateModbusRead+1;
		
	14://read the required registers
		//Start Read Poll 4
		fbMBRead_FC4.nQuantity := usint_Quantity;
		fbMBRead_FC4.nMBAddr := w_Adress;
		fbMBRead_FC4.bExecute := TRUE;
		fbMBRead_FC4.nUnitID := 1;
		timer_Timeout.IN := TRUE;
		IF fbMBRead_FC4.bBusy THEN 
			timer_Delay.IN := TRUE; 
		END_IF
		
		//Wait for Delay, copy Data and then next step
		IF NOT fbMBRead_FC4.bBusy AND NOT fbMBRead_FC4.bError AND timer_Delay.Q THEN
			m_Poll_ok:=TRUE;
			int_Data_Received:=int_Data_Received+1;
			m_MBTCPError := FALSE; 
			
			FOR i:=0 TO 9 BY 1 DO
				arrBuffer_Received[i + WORD_TO_INT(w_Adress)] := arrBuffer_FC4[i];
			END_FOR
			
			//Go to Next Step
			timer_Timeout.IN := FALSE;
			fbMBRead_FC4.bExecute := FALSE;
			timer_Delay.IN := FALSE;		
			iStateModbusRead := iStateModbusRead+1;
		END_IF	

		//Error or Timeout
		IF FPError_FC_4.Q THEN 
			iStateModbusError := 300;
			int_FC4Error := int_FC4Error+1;
		ELSIF timer_Timeout.Q THEN  
			timer_Timeout.IN := FALSE; 	
			iStateModbusError := 300;
			int_TimeoutError := int_TimeoutError+1;
		END_IF
	
	15://Wait and go to next step
		timer_Wait.IN := TRUE;
		
		IF timer_Wait.Q = TRUE THEN
			iStateModbusRead := iStateModbusRead+1;
			timer_Wait.IN :=FALSE;
		END_IF
		
	16: // clean the array  Poll 5
		FOR i:=0 TO 11 BY 1 DO
			arrBuffer_FC4[i] := 0;
		END_FOR
		w_Adress := w_Adress + 10;
		usint_Quantity := 10; 
		iStateModbusRead := iStateModbusRead+1;
		
	17://read the required registers
		//Start Read Poll 5
		fbMBRead_FC4.nQuantity := usint_Quantity;
		fbMBRead_FC4.nMBAddr := w_Adress;
		fbMBRead_FC4.bExecute := TRUE;
		fbMBRead_FC4.nUnitID := 1;
		timer_Timeout.IN := TRUE;
		IF fbMBRead_FC4.bBusy THEN 
			timer_Delay.IN := TRUE; 
		END_IF
		
		//Wait for Delay, copy Data and then next step
		IF NOT fbMBRead_FC4.bBusy AND NOT fbMBRead_FC4.bError AND timer_Delay.Q THEN
			m_Poll_ok:=TRUE;
			int_Data_Received:=int_Data_Received+1;
			m_MBTCPError := FALSE; 
			
			FOR i:=0 TO 9 BY 1 DO
				arrBuffer_Received[i + WORD_TO_INT(w_Adress)] := arrBuffer_FC4[i];
			END_FOR
			
			//Go to Next Step
			timer_Timeout.IN := FALSE;
			fbMBRead_FC4.bExecute := FALSE;
			timer_Delay.IN := FALSE;		
			iStateModbusRead := iStateModbusRead+1;
		END_IF	

		//Error or Timeout
		IF FPError_FC_4.Q THEN 
			iStateModbusError := 300;
			int_FC4Error := int_FC4Error+1;
		ELSIF timer_Timeout.Q THEN  
			timer_Timeout.IN := FALSE; 	
			iStateModbusError := 300;
			int_TimeoutError := int_TimeoutError+1;
		END_IF
	
	18://Wait and go to next step
		timer_Wait.IN := TRUE;
		
		IF timer_Wait.Q = TRUE THEN
			iStateModbusRead := iStateModbusRead+1;
			timer_Wait.IN :=FALSE;
		END_IF	

	19: // clean the array  Poll 6
		FOR i:=0 TO 11 BY 1 DO
			arrBuffer_FC4[i] := 0;
		END_FOR
		w_Adress := w_Adress + 10;
		usint_Quantity := 10; 
		iStateModbusRead := iStateModbusRead+1;
		
	20://read the required registers
		//Start Read Poll 6
		fbMBRead_FC4.nQuantity := usint_Quantity;
		fbMBRead_FC4.nMBAddr := w_Adress;
		fbMBRead_FC4.bExecute := TRUE;
		fbMBRead_FC4.nUnitID := 1;
		timer_Timeout.IN := TRUE;
		IF fbMBRead_FC4.bBusy THEN 
			timer_Delay.IN := TRUE; 
		END_IF
		
		//Wait for Delay, copy Data and then next step
		IF NOT fbMBRead_FC4.bBusy AND NOT fbMBRead_FC4.bError AND timer_Delay.Q THEN
			m_Poll_ok:=TRUE;
			int_Data_Received:=int_Data_Received+1;
			m_MBTCPError := FALSE; 
			
			FOR i:=0 TO 9 BY 1 DO
				arrBuffer_Received[i + WORD_TO_INT(w_Adress)] := arrBuffer_FC4[i];
			END_FOR
			
			//Go to Next Step
			timer_Timeout.IN := FALSE;
			fbMBRead_FC4.bExecute := FALSE;
			timer_Delay.IN := FALSE;		
			iStateModbusRead := iStateModbusRead+1;
		END_IF	

		//Error or Timeout
		IF FPError_FC_4.Q THEN 
			iStateModbusError := 300;
			int_FC4Error := int_FC4Error+1;
		ELSIF timer_Timeout.Q THEN  
			timer_Timeout.IN := FALSE; 	
			iStateModbusError := 300;
			int_TimeoutError := int_TimeoutError+1;
		END_IF
	
	21://Wait and go to next step
		timer_Wait.IN := TRUE;
		
		IF timer_Wait.Q = TRUE THEN
			iStateModbusRead := iStateModbusRead+1;
			timer_Wait.IN :=FALSE;
		END_IF	
		
	22: // clean the array  Poll 7
		FOR i:=0 TO 11 BY 1 DO
			arrBuffer_FC4[i] := 0;
		END_FOR
		w_Adress := w_Adress + 10;
		usint_Quantity := 10; 
		iStateModbusRead := iStateModbusRead+1;
		
	23://read the required registers
		//Start Read Poll 7
		fbMBRead_FC4.nQuantity := usint_Quantity;
		fbMBRead_FC4.nMBAddr := w_Adress;
		fbMBRead_FC4.bExecute := TRUE;
		fbMBRead_FC4.nUnitID := 1;
		timer_Timeout.IN := TRUE;
		IF fbMBRead_FC4.bBusy THEN 
			timer_Delay.IN := TRUE; 
		END_IF
		
		//Wait for Delay, copy Data and then next step
		IF NOT fbMBRead_FC4.bBusy AND NOT fbMBRead_FC4.bError AND timer_Delay.Q THEN
			m_Poll_ok:=TRUE;
			int_Data_Received:=int_Data_Received+1;
			m_MBTCPError := FALSE; 
			
			FOR i:=0 TO 9 BY 1 DO
				arrBuffer_Received[i + WORD_TO_INT(w_Adress)] := arrBuffer_FC4[i];
			END_FOR
			
			//Go to Next Step
			timer_Timeout.IN := FALSE;
			fbMBRead_FC4.bExecute := FALSE;
			timer_Delay.IN := FALSE;		
			iStateModbusRead := iStateModbusRead+1;
		END_IF	

		//Error or Timeout
		IF FPError_FC_4.Q THEN 
			iStateModbusError := 300;
			int_FC4Error := int_FC4Error+1;
		ELSIF timer_Timeout.Q THEN  
			timer_Timeout.IN := FALSE; 	
			iStateModbusError := 300;
			int_TimeoutError := int_TimeoutError+1;
		END_IF
	
	24://Wait and go to next step
		timer_Wait.IN := TRUE;
		
		IF timer_Wait.Q = TRUE THEN
			iStateModbusRead := iStateModbusRead+1;
			timer_Wait.IN :=FALSE;
		END_IF	

	25: // clean the array  Poll 8
		FOR i:=0 TO 11 BY 1 DO
			arrBuffer_FC4[i] := 0;
		END_FOR
		w_Adress := w_Adress + 10;
		usint_Quantity := 10; 
		iStateModbusRead := iStateModbusRead+1;
		
	26://read the required registers
		//Start Read Poll 8
		fbMBRead_FC4.nQuantity := usint_Quantity;
		fbMBRead_FC4.nMBAddr := w_Adress;
		fbMBRead_FC4.bExecute := TRUE;
		fbMBRead_FC4.nUnitID := 1;
		timer_Timeout.IN := TRUE;
		IF fbMBRead_FC4.bBusy THEN 
			timer_Delay.IN := TRUE; 
		END_IF
		
		//Wait for Delay, copy Data and then next step
		IF NOT fbMBRead_FC4.bBusy AND NOT fbMBRead_FC4.bError AND timer_Delay.Q THEN
			m_Poll_ok:=TRUE;
			int_Data_Received:=int_Data_Received+1;
			m_MBTCPError := FALSE; 
			
			FOR i:=0 TO 9 BY 1 DO
				arrBuffer_Received[i + WORD_TO_INT(w_Adress)] := arrBuffer_FC4[i];
			END_FOR
			
			//Go to Next Step
			timer_Timeout.IN := FALSE;
			fbMBRead_FC4.bExecute := FALSE;
			timer_Delay.IN := FALSE;		
			iStateModbusRead := 30;  // convert data
		END_IF	

		//Error or Timeout
		IF FPError_FC_4.Q THEN 
			iStateModbusError := 300;
			int_FC4Error := int_FC4Error+1;
		ELSIF timer_Timeout.Q THEN  
			timer_Timeout.IN := FALSE; 	
			iStateModbusError := 300;
			int_TimeoutError := int_TimeoutError+1;
		END_IF
	
*)
	
	30: // convert data
		real_VoltageL1L2_V 	:= WORD_TO_REAL(arrBuffer_Received[0]) /10;
		real_VoltageL2L3_V 	:= WORD_TO_REAL(arrBuffer_Received[1]) /10;
		real_VoltageL3L1_V 	:= WORD_TO_REAL(arrBuffer_Received[2]) /10;
		real_VoltageL1N_V 	:= WORD_TO_REAL(arrBuffer_Received[4]) /10;
		real_VoltageL2N_V 	:= WORD_TO_REAL(arrBuffer_Received[5]) /10;
		real_VoltageL3N_V 	:= WORD_TO_REAL(arrBuffer_Received[6]) /10;
		real_Frequency_Hz	:= WORD_TO_REAL(arrBuffer_Received[11]) /100;
		
		real_CurrentL1_A	:= WORD_TO_REAL(arrBuffer_Received[100]) /10;
		real_CurrentL2_A	:= WORD_TO_REAL(arrBuffer_Received[101]) /10;
		real_CurrentL3_A	:= WORD_TO_REAL(arrBuffer_Received[102]) /10;
		
		real_RealPowerL1_kW	:= WORD_TO_REAL(arrBuffer_Received[200]) /10;
		real_RealPowerL2_kW	:= WORD_TO_REAL(arrBuffer_Received[201]) /10;
		real_RealPowerL3_kW	:= WORD_TO_REAL(arrBuffer_Received[202]) /10;	
		real_RealPower_kW	:= WORD_TO_REAL(arrBuffer_Received[203]) /10;
		real_ReactivePowerL1_kVAr	:= WORD_TO_REAL(arrBuffer_Received[204]) /10;
		real_ReactivePowerL2_kVAr	:= WORD_TO_REAL(arrBuffer_Received[205]) /10;
		real_ReactivePowerL3_kVAr	:= WORD_TO_REAL(arrBuffer_Received[206]) /10;	
		real_ReactivePower_kVAr	:= WORD_TO_REAL(arrBuffer_Received[207]) /10;
		real_PowerFactorL1	:= WORD_TO_REAL(arrBuffer_Received[208]) /1000;
		real_PowerFactorL2	:= WORD_TO_REAL(arrBuffer_Received[209]) /1000;
		real_PowerFactorL3	:= WORD_TO_REAL(arrBuffer_Received[210]) /1000;	
		real_PowerFactor	:= WORD_TO_REAL(arrBuffer_Received[211]) /1000;

		real_EnergyTotal_Import_kWh		:= WORD_TO_REAL(arrBuffer_Received[301]) /10;
		real_EnergyTotal_Export_kWh		:= WORD_TO_REAL(arrBuffer_Received[303]) /10;
		
		// go to next state
		iStateModbusRead := iStateModbusRead+1;		
		
	31://Wait and go to start
		timer_Wait.IN := TRUE;
		
		IF timer_Wait.Q = TRUE THEN
			iStateModbusRead := 1;
			timer_Wait.IN :=FALSE;
		END_IF	

END_CASE

(* wait timer*)

timer_Wait(PT:=T#1S);


(*------------------------------------------------------------------Error and Warning----------------------------------------------------------------------------*)	
 
timer_Connection_ok			(In:=int_Data_Received<>int_Data_Received_old,PT:=T#10S);
timer_Connection_ok_TOF		(In:=NOT(int_Data_Received<>int_Data_Received_old) AND int_Data_Received>3 ,PT:=T#20S);
int_Data_Received_old:=int_Data_Received;
m_PollSuccessful:=NOT timer_Connection_ok.Q AND timer_Connection_ok_TOF.Q ;

(*------------------------------------------------------------------------------------------Modbus TCP Functions---------------------------------------------------------------------------------------------*)

fbMBRead_FC4(	sIPAddr:= str_IPAdress, 
				nTCPPort:= 502,
				cbLength:= SIZEOF(arrBuffer_FC4), 
				pDestAddr:= ADR(arrBuffer_FC4), 
				tTimeout:= T#10S,
				nErrId => udint_Error_ID);

FPError_FC_4(CLK:= fbMBRead_FC4.bError, Q=> );		

(*------------------------------------------------------------------------------------------State Machine Error---------------------------------------------------------------------------------------------*)	

CASE iStateModbusError OF
	
	300://Error
		timer_Wait.IN :=TRUE;
		timer_Delay.IN := FALSE;
		fbMBRead_FC4.bExecute := FALSE;
		m_MBTCPError := TRUE; 		
		m_Poll_ok:=FALSE;
		int_Data_Received:=0;
		
				//Restart from new with the Read out part after an Error
		IF timer_Wait.Q = TRUE THEN
			iStateModbusRead := 0;	
			iStateModbusError := 0;
			timer_Wait.IN :=FALSE;
			timer_Timeout.IN := FALSE;
		END_IF		
							
END_CASE

END_FUNCTION_BLOCK

// ---- FBs/Huawei/FB_Convert_Huawei_SmartLogger.TcPOU
FUNCTION_BLOCK FB_Convert_Huawei_SmartLogger
VAR_INPUT
	arrBuffer_FC3				: ARRAY[0..25] OF WORD;	
	int_Poll_Counter			:INT;
	
END_VAR
VAR_OUTPUT
	lrPowerTotal			:LREAL;
	lrReactivePowerTotal	:LREAL;
	eOperatingStateInverter	:E_Huawei_SmartLogger_OperatingState;
	
	
END_VAR
VAR
END_VAR

//Copy Data AC Power

lrPowerTotal := DINT_TO_LREAL(SHL(WORD_TO_DWORD(arrBuffer_FC3[0]),16) + WORD_TO_DWORD(arrBuffer_FC3[1]));
lrReactivePowerTotal := DINT_TO_LREAL(SHL(WORD_TO_DWORD(arrBuffer_FC3[2]),16) + WORD_TO_DWORD(arrBuffer_FC3[3]));


//Operating State	
IF 			arrBuffer_FC3[9] = 16#0000 THEN eOperatingStateInverter := 	E_Huawei_SmartLogger_OperatingState.Standby_initializing;
	ELSIF 	arrBuffer_FC3[9] = 16#0001 THEN eOperatingStateInverter := 	E_Huawei_SmartLogger_OperatingState.Standby_detecting_insulation_resistance;
	ELSIF 	arrBuffer_FC3[9] = 16#0002 THEN eOperatingStateInverter := 	E_Huawei_SmartLogger_OperatingState.Standby_detecting_irradiation;
	ELSIF 	arrBuffer_FC3[9] = 16#0003 THEN eOperatingStateInverter := 	E_Huawei_SmartLogger_OperatingState.Standby_gid_detecting;
	ELSIF 	arrBuffer_FC3[9] = 16#0100 THEN eOperatingStateInverter := 	E_Huawei_SmartLogger_OperatingState.Starting;
	ELSIF 	arrBuffer_FC3[9] = 16#0200 THEN eOperatingStateInverter := 	E_Huawei_SmartLogger_OperatingState.On_grid_Off_grid_mode_running;
	ELSIF 	arrBuffer_FC3[9] = 16#0201 THEN eOperatingStateInverter := 	E_Huawei_SmartLogger_OperatingState.Grid_connection_power_limited_Off_mode_running_power_limited;
	ELSIF 	arrBuffer_FC3[9] = 16#0202 THEN eOperatingStateInverter := 	E_Huawei_SmartLogger_OperatingState.Grid_connection_selfderating_Off_mode_running_selfderating;
	ELSIF 	arrBuffer_FC3[9] = 16#0203 THEN eOperatingStateInverter := 	E_Huawei_SmartLogger_OperatingState.Off_grid_Running;
	ELSIF 	arrBuffer_FC3[9] = 16#0300 THEN eOperatingStateInverter := 	E_Huawei_SmartLogger_OperatingState.Shutdown_fault;
	ELSIF 	arrBuffer_FC3[9] = 16#0301 THEN eOperatingStateInverter := 	E_Huawei_SmartLogger_OperatingState.Shutdown_command;
	ELSIF 	arrBuffer_FC3[9] = 16#0302 THEN eOperatingStateInverter := 	E_Huawei_SmartLogger_OperatingState.Shutdown_OVGR;
	ELSIF 	arrBuffer_FC3[9] = 16#0303 THEN eOperatingStateInverter := 	E_Huawei_SmartLogger_OperatingState.Shutdown_communication_disconnected;
	ELSIF 	arrBuffer_FC3[9] = 16#0304 THEN eOperatingStateInverter := 	E_Huawei_SmartLogger_OperatingState.Shutdown_power_limited	;
	ELSIF 	arrBuffer_FC3[9] = 16#0305 THEN eOperatingStateInverter := 	E_Huawei_SmartLogger_OperatingState.Shutdown_manual_startup_required;
	ELSIF 	arrBuffer_FC3[9] = 16#0306 THEN eOperatingStateInverter := 	E_Huawei_SmartLogger_OperatingState.Shutdown_DC_switches_disconnected;
	ELSIF 	arrBuffer_FC3[9] = 16#0307 THEN eOperatingStateInverter := 	E_Huawei_SmartLogger_OperatingState.Shutdown_rapid_cutoff;
	ELSIF 	arrBuffer_FC3[9] = 16#0308 THEN eOperatingStateInverter := 	E_Huawei_SmartLogger_OperatingState.Shutdown_input_underpower;
	ELSIF 	arrBuffer_FC3[9] = 16#0401 THEN eOperatingStateInverter := 	E_Huawei_SmartLogger_OperatingState.Grid_scheduling_cosphi_P_curve;
	ELSIF 	arrBuffer_FC3[9] = 16#0402 THEN eOperatingStateInverter := 	E_Huawei_SmartLogger_OperatingState.Grid_scheduling_Q_U_curve;
	ELSIF 	arrBuffer_FC3[9] = 16#0403 THEN eOperatingStateInverter := 	E_Huawei_SmartLogger_OperatingState.Grid_scheduling_PF_U_curve;
	ELSIF 	arrBuffer_FC3[9] = 16#0404 THEN eOperatingStateInverter := 	E_Huawei_SmartLogger_OperatingState.Grid_scheduling_dry_contact;
	ELSIF 	arrBuffer_FC3[9] = 16#0405 THEN eOperatingStateInverter := 	E_Huawei_SmartLogger_OperatingState.Grid_scheduling_Q_P_curve;
	ELSIF 	arrBuffer_FC3[9] = 16#0500 THEN eOperatingStateInverter := 	E_Huawei_SmartLogger_OperatingState.Spotcheck_ready	;
	ELSIF 	arrBuffer_FC3[9] = 16#0501 THEN eOperatingStateInverter := 	E_Huawei_SmartLogger_OperatingState.Spotchecking;
	ELSIF 	arrBuffer_FC3[9] = 16#0600 THEN eOperatingStateInverter := 	E_Huawei_SmartLogger_OperatingState.Inspecting;
	ELSIF 	arrBuffer_FC3[9] = 16#0700 THEN eOperatingStateInverter := 	E_Huawei_SmartLogger_OperatingState.AFCI_self_check;
	ELSIF 	arrBuffer_FC3[9] = 16#0800 THEN eOperatingStateInverter := 	E_Huawei_SmartLogger_OperatingState.I_V_scanning;
	ELSIF 	arrBuffer_FC3[9] = 16#0900 THEN eOperatingStateInverter := 	E_Huawei_SmartLogger_OperatingState.DC_input_detection;
	ELSIF 	arrBuffer_FC3[9] = 16#0A00 THEN eOperatingStateInverter := 	E_Huawei_SmartLogger_OperatingState.Running_off_grid_charging;
	ELSIF 	arrBuffer_FC3[9] = 16#A000 THEN eOperatingStateInverter := 	E_Huawei_SmartLogger_OperatingState.Standby_no_irradiation;
	ELSIF 	arrBuffer_FC3[9] = 16#B000 THEN eOperatingStateInverter := 	E_Huawei_SmartLogger_OperatingState.Communication_interrupt	;
	ELSIF 	arrBuffer_FC3[9] = 16#C000 THEN eOperatingStateInverter := 	E_Huawei_SmartLogger_OperatingState.Uploading;
	ELSE 									eOperatingStateInverter := 	E_Huawei_SmartLogger_OperatingState.Unknown;
END_IF

	(*	0x0000 Standby: initializing
		0x0001 Standby: detecting insulation resistance
		0x0002 Standby: detecting irradiation
		0x0003 Standby: drid detecting
		0x0100 Starting
		0x0200 On-grid (Off-grid mode: running)
		0x0201 Grid connection: power limited (Off mode: running: power limited)
		0x0202 Grid connection: selfderating (Off mode: running: selfderating)
		0x0203 Off-grid Running
		0x0300 Shutdown: fault
		0x0301 Shutdown: command
		0x0302 Shutdown: OVGR
		0x0303 Shutdown: communication disconnected
		0x0304 Shutdown: power limited
		0x0305 Shutdown: manual startup required
		0x0306 Shutdown: DC switches disconnected
		0x0307 Shutdown: rapid cutoff
		0x0308 Shutdown: input underpower
		0x0401 Grid scheduling: cosφ-P curve
		0x0402 Grid scheduling: Q-U curve
		0x0403 Grid scheduling: PF-U curve
		0x0404 Grid scheduling: dry contact
		0x0405 Grid scheduling: Q-P curve
		0x0500 Spotcheck ready
		0x0501 Spotchecking
		0x0600 Inspecting
		0X0700 AFCI self check
		0X0800 I-V scanning
		0X0900 DC input detection
		0X0A00 Running: off-grid charging
		0xA000 Standby: no irradiation	
		0xB000	Communication interrupt
		0xC000	Uploading					*)

END_FUNCTION_BLOCK

// ---- FBs/Huawei/FB_Huawei_SmartLogger.TcPOU
// {attribute 'hide_all_locals'}
FUNCTION_BLOCK FB_Huawei_SmartLogger
VAR_INPUT PERSISTENT
	bEnable						: BOOL;				//True = Function is enabled, FALSE = Function is dissabled, no new Data
	sIPAdress					: STRING(15);		//IP Adress from the Inverter
	sint_ID_Iverter1			:SINT;				// ID of inveter 1
	sint_ID_Iverter2			:SINT;				// ID of inveter 2
	sint_ID_Iverter3			:SINT;				// ID of inveter 3
	sint_ID_Iverter4			:SINT;				// ID of inveter 4
	sint_ID_Iverter5			:SINT;				// ID of inveter 5
	sint_ID_Iverter6			:SINT;				// ID of inveter 6
	sint_ID_Iverter7			:SINT;				// ID of inveter 7
	sint_ID_Iverter8			:SINT;				// ID of inveter 8
	sint_ID_Iverter9			:SINT;				// ID of inveter 9
	sint_ID_Iverter10			:SINT;				// ID of inveter 10
	sint_ID_Iverter11			:SINT;				// ID of inveter 11
	sint_ID_Iverter12			:SINT;				// ID of inveter 12
	
	
END_VAR
VAR_OUTPUT
	st_Huawei_SmartLogger		: ARRAY[1..20] OF ST_Huawei_SmartLogger_OutData;					//Output structure with Data 
	stDataEMPower_PV			: ARRAY[1..20] OF ST_ElectricMeter_Output_Power;					//Output structure with Data from Electric Meter PV (Power Data)
	stDataEMCounter_PV 			: ARRAY[1..20] OF ST_ElectricMeter_Output_Counter;					//Output structure with Data from Electric Meter PV (Counter Data)
	diNrOfEM_OUT_PV				: DINT;																//Active Number from the Electric Meter for using on other functions
END_VAR
VAR
	sint_ID_Iverter				:ARRAY[1..12] OF SINT;				// Array of ID of inveter 
	fbMeter						: ARRAY[1..30] OF FB_ElectricMeter;					//Electric Meter Function 
	fbElMeter					: FB_ElectricMeter;									//Electric Meter Function for sumation values 
	
	fbNumberDevice				: FB_NumberOfDevice;								//Function block to calcualte the number of the Device
	fbConvertEnergyRegister		: FB_CV_WORD_TO_DWORD;								//Convert function
	fbMBRead_FC3				: FB_MBReadRegs;									//Modbus Read Function (FC3)
	timDelay					: TON;												//Timer for Delay between Requests
	timTimeout					: TON;												//Timer for Timeout
	timDissableFunctions		: TON;												//Timer to dissable the Function after Lynus_Standards.Constants_General.tTimeDissableLynusFunctions Days without connection to the Lynus Cloud
	timResetConnectionOnGVL		: TON;												//Timer to try reset the connection Flag on the GVL. (When somebody delete the Connection Function and make only a onlinechange)
	FPEnable					: R_TRIG;											//Internal positive Edge
	FPError_FC_3				: R_TRIG;											//Internal positive Edge
	PD_String					: FB_PersistentData_String;							//Function to save persistent data 
	stFloat						: ST_UN_FLOAT_CONVERT_DWORD_REAL;					//Convert the Float Raw Value
	arrBuffer_FC3				: ARRAY[0..25] OF WORD;							//Buffer with Data from FC3
	arrPD						: ARRAY[1..2] OF FB_PersistentData_Number;			//Function to save persistent data 
	byWaitInStep				: BYTE;												//Wait in Step before start to clean data on PLC
	iStateGVLData				: INT;												//State machine to handle the data on the GVL
	iStateModbus				: INT;												//State variable for Statemachine
	iStateModbus_CP				: INT;												//Compare State variable
	diCounterForGVL				: DINT;												//Counter to clean old data on GVL
	lrCheckValue				: LREAL;											//Internal Value to check the value before convert
	x							: INT;
	i: INT;
	int_Poll_Counter			: INT;												//Poll1 = inverter_ID 1,....
	byLPForInverter: INT;
	lrCounterEnergyProduction: LREAL;
	dwInput: DWORD;
	int_maxPolls				:INT :=12;											//maximum number of polls / inverter. 
	ton_Wait: Ton;
	FB_ConvertData			:FB_Convert_Huawei_SmartLogger;
	lreal1: LREAL;
	lreal2: LREAL;
	lreal3: LREAL;
	lreal4: LREAL;
	lreal5: LREAL;
	lreal6: LREAL;
	lreal7: LREAL;
	lreal8: LREAL;
	lreal9: LREAL;
	lreal10: LREAL;
	lreal11: LREAL;
	lreal12: LREAL;
	lreal13: LREAL;
	lreal14: LREAL;
	lreal15: LREAL;
	lreal16: LREAL;
	lreal17: LREAL;
	lreal18: LREAL;
	lreal19: LREAL;
	lreal20: LREAL;
	END_VAR

//Creator : Stefan Lackner
//Company : EfficientIO
//Date : 17.10.2022
//Version : 0.0.0.1		

//With this function its possible to read out values from the SmartLogger from the manufacturer Huawei
//This Function read out the Values from up to 12 inverters behind a SmartLogger. The SmartLogger could handle up to 247 inverters. 
//The protocol to the Inverter is Modbus TCP
//Attention. To access the registers, an offset of 1 must always be subtracted. Register 40001 would then be on register 40000.
//The document "SmartLogger ModBus Interface Definitions.pdf" issue 35 got used for the Modbus adress List

//NOTE for diNr.....Designation => 
//_IN = Here Data come in from other Functions or go out to other functions about the GVL
//_OUT = Here Data go out to other functions about the GVL


(*------------------------------------------------------------------------------------------General Input Part---------------------------------------------------------------------------------------------*)

//Check limitation
sint_ID_Iverter1 := LIMIT(0,sint_ID_Iverter1,127);
sint_ID_Iverter2 := LIMIT(0,sint_ID_Iverter2,127);
sint_ID_Iverter3 := LIMIT(0,sint_ID_Iverter3,127);
sint_ID_Iverter4 := LIMIT(0,sint_ID_Iverter4,127);
sint_ID_Iverter5 := LIMIT(0,sint_ID_Iverter5,127);
sint_ID_Iverter6 := LIMIT(0,sint_ID_Iverter6,127);
sint_ID_Iverter7 := LIMIT(0,sint_ID_Iverter7,127);
sint_ID_Iverter8 := LIMIT(0,sint_ID_Iverter8,127);
sint_ID_Iverter9 := LIMIT(0,sint_ID_Iverter9,127);
sint_ID_Iverter10:= LIMIT(0,sint_ID_Iverter10,127);
sint_ID_Iverter11:= LIMIT(0,sint_ID_Iverter11,127);
sint_ID_Iverter12 := LIMIT(0,sint_ID_Iverter12,127);
// copy in an array, easier for handling in the state maschine
sint_ID_Iverter[1]	:=	sint_ID_Iverter1;
sint_ID_Iverter[2]	:=	sint_ID_Iverter2;
sint_ID_Iverter[3]	:=	sint_ID_Iverter3;
sint_ID_Iverter[4]	:=	sint_ID_Iverter4;
sint_ID_Iverter[5]	:=	sint_ID_Iverter5;
sint_ID_Iverter[6]	:=	sint_ID_Iverter6;
sint_ID_Iverter[7]	:=	sint_ID_Iverter7;
sint_ID_Iverter[8]	:=	sint_ID_Iverter8;
sint_ID_Iverter[9]	:=	sint_ID_Iverter9;
sint_ID_Iverter[10]	:=	sint_ID_Iverter10;
sint_ID_Iverter[11]	:=	sint_ID_Iverter11;
sint_ID_Iverter[12]	:=	sint_ID_Iverter12;



(*-------------------------------------------------------------Calcualte the number of EM System---------------------------------------------------------------*)

fbNumberDevice(
	diActualNumberOfDevices:= Lynus_Standards.GVL_Energy.stNumberOfDevices.diNumberOfElectricMeters, 
	diMaxNumberOfDevices:= Constants_Energy.diMaxNumberOfElectricMeters, 
	udiCounterOnlineChange:= TwinCAT_SystemInfoVarList._AppInfo.OnlineChangeCnt, 
	bNumberIsCalculatet=> , 
	bFPNumberIsCalculatet=> , 
	bOnlineChange=> , 
	diNumberForThisDevice=> diNrOfEM_OUT_PV, 
	diNumberOfTotalDevices=> );

//Write new Numer on GVL
IF fbNumberDevice.bFPNumberIsCalculatet THEN
	Lynus_Standards.GVL_Energy.stNumberOfDevices.diNumberOfElectricMeters := fbNumberDevice.diNumberOfTotalDevices;	
END_IF 

//Delete old Number on GVL
IF fbNumberDevice.bOnlineChange THEN 
	Lynus_Standards.GVL_Energy.stNumberOfDevices.diNumberOfElectricMeters := diNrOfEM_OUT_PV;	
		iStateGVLData := 1; 
END_IF

(*-------------------------------------------------------------Service from Backend is ready and check the connection to backend for dissabel/enable Function---------------------------------------------------------------*)

//Try to reset the variable for connection on the GVL. When all is normal then the EfficientIO Mqtt connection function set this variable to true in the next cycle
//When we have no connection to the backend then after Lynus_Standards.Constants_General.tTimeDissableLynusFunctions days the Function is dissabled with all of his functionalities
timResetConnectionOnGVL(IN:= NOT timResetConnectionOnGVL.Q, PT:= T#1H, Q=> , ET=> );
IF timResetConnectionOnGVL.Q THEN 
	Lynus_Standards.GVL_Communicator.bStateConnectionToEnableFunctions := FALSE; 
END_IF
IF NOT Lynus_Standards.GVL_Communicator.bStateConnectionToEnableFunctions THEN 
	timDissableFunctions.IN := TRUE; 
ELSE 
	timDissableFunctions.IN := FALSE; 
END_IF  
timDissableFunctions(IN:= , PT:= Lynus_Standards.Constants_General.tTimeDissableLynusFunctions, Q=> , ET=> );
	
(*------------------------------------------------------------------------------------------State Machine---------------------------------------------------------------------------------------------*)
	
//Enable
FPEnable(CLK:= bEnable, Q=> );
IF FPEnable.Q AND iStateModbus = 0 THEN 
	iStateModbus := 1; 
END_IF
IF NOT bEnable OR timDissableFunctions.Q THEN 
	iStateModbus := 0; 
END_IF

//Timer for delay
timDelay(IN:= , PT:= T#100MS, Q=> , ET=> );	

//Timer for Timeout in Statemachine
IF iStateModbus = iStateModbus_CP THEN 
	timTimeout.IN := TRUE; 
ELSE 
	timTimeout.IN := FALSE; 
END_IF
IF iStateModbus = 0 THEN 
	timTimeout.IN := FALSE; 
END_IF
timTimeout(IN:= , PT:= T#20S, Q=> , ET=> );	


//Statemachine
CASE iStateModbus OF
	
	0://Init Step
		iStateModbus_CP := iStateModbus;
		timDelay.IN := FALSE;
		FOR i:=1 TO 20 BY 1 DO
			st_Huawei_SmartLogger[i].bFunctionIsActive := FALSE;
			st_Huawei_SmartLogger[i].eOperatingStateInverter := E_Huawei_SmartLogger_OperatingState.Unknown ;
		END_FOR
		
		fbMBRead_FC3.bExecute := FALSE;
		lrCheckValue := 0;
									
	1://Read out first inverter
		int_Poll_Counter:=1;			//Poll int_Poll_Counter : Inverter int_Poll_Counter 	
		st_Huawei_SmartLogger[int_Poll_Counter].bFunctionIsActive := TRUE;
		iStateModbus_CP := iStateModbus;
		fbMBRead_FC3.nQuantity := 25;
		fbMBRead_FC3.nMBAddr := (51000+(25*(SINT_TO_WORD(sint_ID_Iverter[int_Poll_Counter]) - 1)));
		fbMBRead_FC3.bExecute := TRUE;
			
		IF fbMBRead_FC3.bBusy THEN 
			timDelay.IN := TRUE; 
		END_IF
		
		//Wait for Delay, copy Data and then next step
		IF NOT fbMBRead_FC3.bBusy AND NOT fbMBRead_FC3.bError AND timDelay.Q THEN
			// convert received data
			FB_ConvertData(	arrBuffer_FC3			:=	arrBuffer_FC3,
											int_Poll_Counter		:=	int_Poll_Counter,
											lrPowerTotal			=>	fbMeter[int_Poll_Counter].lrPowerTotal,	
											lrReactivePowerTotal	=> 	fbMeter[int_Poll_Counter].lrReactivePowerTotal,
											eOperatingStateInverter	=>	st_Huawei_SmartLogger[int_Poll_Counter].eOperatingStateInverter);
	
			//Next Step
			fbMBRead_FC3.bExecute := FALSE;
			timDelay.IN := FALSE;
			iStateModbus := iStateModbus+1;
			IF arrBuffer_FC3[9]<>0 THEN
				st_Huawei_SmartLogger[int_Poll_Counter].bError := FALSE; 
				st_Huawei_SmartLogger[int_Poll_Counter].eErrorState := E_Huawei_SmartLogger_Error.eNoError;
			ELSE
				st_Huawei_SmartLogger[int_Poll_Counter].bError := FALSE; 
				st_Huawei_SmartLogger[int_Poll_Counter].eErrorState := E_Huawei_SmartLogger_Error.eNoError;
			END_IF
		END_IF
			
		//Error from Inverter 
		IF NOT fbMBRead_FC3.bBusy AND NOT fbMBRead_FC3.bError AND timDelay.Q AND arrBuffer_FC3[9] >= 16#0300 AND arrBuffer_FC3[9] <= 16#0308 THEN
			iStateModbus := 300;
			st_Huawei_SmartLogger[int_Poll_Counter].eErrorState := E_Huawei_SmartLogger_Error.eHuawei_SmartLoggerError;
		END_IF
	
		//Error or Timeout
		IF FPError_FC_3.Q OR timTimeout.Q THEN
			iStateModbus := 300;
			st_Huawei_SmartLogger[int_Poll_Counter].eOperatingStateInverter := E_Huawei_SmartLogger_OperatingState.Unknown;
			st_Huawei_SmartLogger[int_Poll_Counter].eErrorState	:=	E_Huawei_SmartLogger_Error.eModbusTCPError;
		END_IF
		
	2://Wait and go to step 1 or step 3
		iStateModbus_CP := iStateModbus;
		IF sint_ID_Iverter[int_Poll_Counter+1] = 0 OR int_Poll_Counter=int_maxPolls THEN		// if ID is not in use, go to state 100
			iStateModbus := 100;
		ELSE
			iStateModbus := 3;
			int_Poll_Counter:=int_Poll_Counter+1;			//Poll int_Poll_Counter : Inverter int_Poll_Counter 	
		END_IF

	3://Read out next inverter
		st_Huawei_SmartLogger[int_Poll_Counter].bFunctionIsActive := TRUE;
		iStateModbus_CP := iStateModbus;
		fbMBRead_FC3.nQuantity := 25;
		fbMBRead_FC3.nMBAddr := (51000+(25*(SINT_TO_WORD(sint_ID_Iverter[int_Poll_Counter]) - 1)));
		fbMBRead_FC3.bExecute := TRUE;
			
		IF fbMBRead_FC3.bBusy THEN 
			timDelay.IN := TRUE; 
		END_IF
		
		//Wait for Delay, copy Data and then next step
		IF NOT fbMBRead_FC3.bBusy AND NOT fbMBRead_FC3.bError AND timDelay.Q THEN
			// convert received data
			FB_ConvertData(	arrBuffer_FC3			:=	arrBuffer_FC3,
											int_Poll_Counter		:=	int_Poll_Counter,
											lrPowerTotal			=>	fbMeter[int_Poll_Counter].lrPowerTotal,	
											lrReactivePowerTotal	=> 	fbMeter[int_Poll_Counter].lrReactivePowerTotal,
											eOperatingStateInverter	=>	st_Huawei_SmartLogger[int_Poll_Counter].eOperatingStateInverter);
	
			//Next Step
			fbMBRead_FC3.bExecute := FALSE;
			timDelay.IN := FALSE;
			iStateModbus := iStateModbus+1;
			IF arrBuffer_FC3[9]<>0 THEN
				st_Huawei_SmartLogger[int_Poll_Counter].bError := FALSE; 
				st_Huawei_SmartLogger[int_Poll_Counter].eErrorState := E_Huawei_SmartLogger_Error.eNoError;
			ELSE
				st_Huawei_SmartLogger[int_Poll_Counter].bError := FALSE; 
				st_Huawei_SmartLogger[int_Poll_Counter].eErrorState := E_Huawei_SmartLogger_Error.eNoError;
			END_IF
		END_IF
			
		//Error from Inverter 
		IF NOT fbMBRead_FC3.bBusy AND NOT fbMBRead_FC3.bError AND timDelay.Q AND arrBuffer_FC3[9] >= 16#0300 AND arrBuffer_FC3[9] <= 16#0308 THEN
			iStateModbus := 300;
			st_Huawei_SmartLogger[int_Poll_Counter].eErrorState := E_Huawei_SmartLogger_Error.eHuawei_SmartLoggerError;
		END_IF
	
		//Error or Timeout
		IF FPError_FC_3.Q OR timTimeout.Q THEN
			iStateModbus := 300;
			st_Huawei_SmartLogger[int_Poll_Counter].eOperatingStateInverter := E_Huawei_SmartLogger_OperatingState.Unknown;
			st_Huawei_SmartLogger[int_Poll_Counter].eErrorState	:=	E_Huawei_SmartLogger_Error.eModbusTCPError;
		END_IF
		
	4://Wait and go to step +1 or step 100
		iStateModbus_CP := iStateModbus;
		IF sint_ID_Iverter[int_Poll_Counter+1] = 0 OR int_Poll_Counter=int_maxPolls THEN		// if ID is not in use, go to state 100
			iStateModbus := 100;
		ELSE
			iStateModbus := iStateModbus+1;
			int_Poll_Counter:=int_Poll_Counter+1;			//Poll int_Poll_Counter : Inverter int_Poll_Counter 	
		END_IF
	
	5://Read out next inverter
		st_Huawei_SmartLogger[int_Poll_Counter].bFunctionIsActive := TRUE;
		iStateModbus_CP := iStateModbus;
		fbMBRead_FC3.nQuantity := 25;
		fbMBRead_FC3.nMBAddr := (51000+(25*(SINT_TO_WORD(sint_ID_Iverter[int_Poll_Counter]) - 1)));
		fbMBRead_FC3.bExecute := TRUE;
			
		IF fbMBRead_FC3.bBusy THEN 
			timDelay.IN := TRUE; 
		END_IF
		
		//Wait for Delay, copy Data and then next step
		IF NOT fbMBRead_FC3.bBusy AND NOT fbMBRead_FC3.bError AND timDelay.Q THEN
			// convert received data
			FB_ConvertData(	arrBuffer_FC3			:=	arrBuffer_FC3,
											int_Poll_Counter		:=	int_Poll_Counter,
											lrPowerTotal			=>	fbMeter[int_Poll_Counter].lrPowerTotal,	
											lrReactivePowerTotal	=> 	fbMeter[int_Poll_Counter].lrReactivePowerTotal,
											eOperatingStateInverter	=>	st_Huawei_SmartLogger[int_Poll_Counter].eOperatingStateInverter);
	
			//Next Step
			fbMBRead_FC3.bExecute := FALSE;
			timDelay.IN := FALSE;
			iStateModbus := iStateModbus+1;
			IF arrBuffer_FC3[9]<>0 THEN
				st_Huawei_SmartLogger[int_Poll_Counter].bError := FALSE; 
				st_Huawei_SmartLogger[int_Poll_Counter].eErrorState := E_Huawei_SmartLogger_Error.eNoError;
			ELSE
				st_Huawei_SmartLogger[int_Poll_Counter].bError := FALSE; 
				st_Huawei_SmartLogger[int_Poll_Counter].eErrorState := E_Huawei_SmartLogger_Error.eNoError;
			END_IF
		END_IF
			
		//Error from Inverter 
		IF NOT fbMBRead_FC3.bBusy AND NOT fbMBRead_FC3.bError AND timDelay.Q AND arrBuffer_FC3[9] >= 16#0300 AND arrBuffer_FC3[9] <= 16#0308 THEN
			iStateModbus := 300;
			st_Huawei_SmartLogger[int_Poll_Counter].eErrorState := E_Huawei_SmartLogger_Error.eHuawei_SmartLoggerError;
		END_IF
	
		//Error or Timeout
		IF FPError_FC_3.Q OR timTimeout.Q THEN
			iStateModbus := 300;
			st_Huawei_SmartLogger[int_Poll_Counter].eOperatingStateInverter := E_Huawei_SmartLogger_OperatingState.Unknown;
			st_Huawei_SmartLogger[int_Poll_Counter].eErrorState	:=	E_Huawei_SmartLogger_Error.eModbusTCPError;
		END_IF
		
	6://Wait and go to step +1 or step 100
		iStateModbus_CP := iStateModbus;
		IF sint_ID_Iverter[int_Poll_Counter+1] = 0 OR int_Poll_Counter=int_maxPolls THEN		// if ID is not in use, go to state 100
			iStateModbus := 100;
		ELSE
			iStateModbus := iStateModbus+1;
			int_Poll_Counter:=int_Poll_Counter+1;			//Poll int_Poll_Counter : Inverter int_Poll_Counter 	
		END_IF
		
	7://Read out next inverter
		st_Huawei_SmartLogger[int_Poll_Counter].bFunctionIsActive := TRUE;
		iStateModbus_CP := iStateModbus;
		fbMBRead_FC3.nQuantity := 25;
		fbMBRead_FC3.nMBAddr := (51000+(25*(SINT_TO_WORD(sint_ID_Iverter[int_Poll_Counter]) - 1)));
		fbMBRead_FC3.bExecute := TRUE;
			
		IF fbMBRead_FC3.bBusy THEN 
			timDelay.IN := TRUE; 
		END_IF
		
		//Wait for Delay, copy Data and then next step
		IF NOT fbMBRead_FC3.bBusy AND NOT fbMBRead_FC3.bError AND timDelay.Q THEN
			// convert received data
			FB_ConvertData(	arrBuffer_FC3			:=	arrBuffer_FC3,
											int_Poll_Counter		:=	int_Poll_Counter,
											lrPowerTotal			=>	fbMeter[int_Poll_Counter].lrPowerTotal,	
											lrReactivePowerTotal	=> 	fbMeter[int_Poll_Counter].lrReactivePowerTotal,
											eOperatingStateInverter	=>	st_Huawei_SmartLogger[int_Poll_Counter].eOperatingStateInverter);
	
			//Next Step
			fbMBRead_FC3.bExecute := FALSE;
			timDelay.IN := FALSE;
			iStateModbus := iStateModbus+1;
			IF arrBuffer_FC3[9]<>0 THEN
				st_Huawei_SmartLogger[int_Poll_Counter].bError := FALSE; 
				st_Huawei_SmartLogger[int_Poll_Counter].eErrorState := E_Huawei_SmartLogger_Error.eNoError;
			ELSE
				st_Huawei_SmartLogger[int_Poll_Counter].bError := FALSE; 
				st_Huawei_SmartLogger[int_Poll_Counter].eErrorState := E_Huawei_SmartLogger_Error.eNoError;
			END_IF
		END_IF
			
		//Error from Inverter 
		IF NOT fbMBRead_FC3.bBusy AND NOT fbMBRead_FC3.bError AND timDelay.Q AND arrBuffer_FC3[9] >= 16#0300 AND arrBuffer_FC3[9] <= 16#0308 THEN
			iStateModbus := 300;
			st_Huawei_SmartLogger[int_Poll_Counter].eErrorState := E_Huawei_SmartLogger_Error.eHuawei_SmartLoggerError;
		END_IF
	
		//Error or Timeout
		IF FPError_FC_3.Q OR timTimeout.Q THEN
			iStateModbus := 300;
			st_Huawei_SmartLogger[int_Poll_Counter].eOperatingStateInverter := E_Huawei_SmartLogger_OperatingState.Unknown;
			st_Huawei_SmartLogger[int_Poll_Counter].eErrorState	:=	E_Huawei_SmartLogger_Error.eModbusTCPError;
		END_IF

	8://Wait and go to step +1 or step 100
		iStateModbus_CP := iStateModbus;
		IF sint_ID_Iverter[int_Poll_Counter+1] = 0 OR int_Poll_Counter=int_maxPolls THEN		// if ID is not in use, go to state 100
			iStateModbus := 100;
		ELSE
			iStateModbus := iStateModbus+1;
			int_Poll_Counter:=int_Poll_Counter+1;			//Poll int_Poll_Counter : Inverter int_Poll_Counter 	
		END_IF
		
	9://Read out next inverter
		st_Huawei_SmartLogger[int_Poll_Counter].bFunctionIsActive := TRUE;
		iStateModbus_CP := iStateModbus;
		fbMBRead_FC3.nQuantity := 25;
		fbMBRead_FC3.nMBAddr := (51000+(25*(SINT_TO_WORD(sint_ID_Iverter[int_Poll_Counter]) - 1)));
		fbMBRead_FC3.bExecute := TRUE;
			
		IF fbMBRead_FC3.bBusy THEN 
			timDelay.IN := TRUE; 
		END_IF
		
		//Wait for Delay, copy Data and then next step
		IF NOT fbMBRead_FC3.bBusy AND NOT fbMBRead_FC3.bError AND timDelay.Q THEN
			// convert received data
			FB_ConvertData(	arrBuffer_FC3			:=	arrBuffer_FC3,
											int_Poll_Counter		:=	int_Poll_Counter,
											lrPowerTotal			=>	fbMeter[int_Poll_Counter].lrPowerTotal,	
											lrReactivePowerTotal	=> 	fbMeter[int_Poll_Counter].lrReactivePowerTotal,
											eOperatingStateInverter	=>	st_Huawei_SmartLogger[int_Poll_Counter].eOperatingStateInverter);
	
			//Next Step
			fbMBRead_FC3.bExecute := FALSE;
			timDelay.IN := FALSE;
			iStateModbus := iStateModbus+1;
			IF arrBuffer_FC3[9]<>0 THEN
				st_Huawei_SmartLogger[int_Poll_Counter].bError := FALSE; 
				st_Huawei_SmartLogger[int_Poll_Counter].eErrorState := E_Huawei_SmartLogger_Error.eNoError;
			ELSE
				st_Huawei_SmartLogger[int_Poll_Counter].bError := FALSE; 
				st_Huawei_SmartLogger[int_Poll_Counter].eErrorState := E_Huawei_SmartLogger_Error.eNoError;
			END_IF
		END_IF
			
		//Error from Inverter 
		IF NOT fbMBRead_FC3.bBusy AND NOT fbMBRead_FC3.bError AND timDelay.Q AND arrBuffer_FC3[9] >= 16#0300 AND arrBuffer_FC3[9] <= 16#0308 THEN
			iStateModbus := 300;
			st_Huawei_SmartLogger[int_Poll_Counter].eErrorState := E_Huawei_SmartLogger_Error.eHuawei_SmartLoggerError;
		END_IF
	
		//Error or Timeout
		IF FPError_FC_3.Q OR timTimeout.Q THEN
			iStateModbus := 300;
			st_Huawei_SmartLogger[int_Poll_Counter].eOperatingStateInverter := E_Huawei_SmartLogger_OperatingState.Unknown;
			st_Huawei_SmartLogger[int_Poll_Counter].eErrorState	:=	E_Huawei_SmartLogger_Error.eModbusTCPError;
		END_IF
		
	10://Wait and go to step +1 or step 100
		iStateModbus_CP := iStateModbus;
		IF sint_ID_Iverter[int_Poll_Counter+1] = 0 OR int_Poll_Counter=int_maxPolls THEN		// if ID is not in use, go to state 100
			iStateModbus := 100;
		ELSE
			iStateModbus := iStateModbus+1;
			int_Poll_Counter:=int_Poll_Counter+1;			//Poll int_Poll_Counter : Inverter int_Poll_Counter 	
		END_IF
		
	11://Read out next inverter
		st_Huawei_SmartLogger[int_Poll_Counter].bFunctionIsActive := TRUE;
		iStateModbus_CP := iStateModbus;
		fbMBRead_FC3.nQuantity := 25;
		fbMBRead_FC3.nMBAddr := (51000+(25*(SINT_TO_WORD(sint_ID_Iverter[int_Poll_Counter]) - 1)));
		fbMBRead_FC3.bExecute := TRUE;
			
		IF fbMBRead_FC3.bBusy THEN 
			timDelay.IN := TRUE; 
		END_IF
		
		//Wait for Delay, copy Data and then next step
		IF NOT fbMBRead_FC3.bBusy AND NOT fbMBRead_FC3.bError AND timDelay.Q THEN
			// convert received data
			FB_ConvertData(	arrBuffer_FC3			:=	arrBuffer_FC3,
											int_Poll_Counter		:=	int_Poll_Counter,
											lrPowerTotal			=>	fbMeter[int_Poll_Counter].lrPowerTotal,	
											lrReactivePowerTotal	=> 	fbMeter[int_Poll_Counter].lrReactivePowerTotal,
											eOperatingStateInverter	=>	st_Huawei_SmartLogger[int_Poll_Counter].eOperatingStateInverter);
	
			//Next Step
			fbMBRead_FC3.bExecute := FALSE;
			timDelay.IN := FALSE;
			iStateModbus := iStateModbus+1;
			IF arrBuffer_FC3[9]<>0 THEN
				st_Huawei_SmartLogger[int_Poll_Counter].bError := FALSE; 
				st_Huawei_SmartLogger[int_Poll_Counter].eErrorState := E_Huawei_SmartLogger_Error.eNoError;
			ELSE
				st_Huawei_SmartLogger[int_Poll_Counter].bError := FALSE; 
				st_Huawei_SmartLogger[int_Poll_Counter].eErrorState := E_Huawei_SmartLogger_Error.eNoError;
			END_IF
		END_IF
			
		//Error from Inverter 
		IF NOT fbMBRead_FC3.bBusy AND NOT fbMBRead_FC3.bError AND timDelay.Q AND arrBuffer_FC3[9] >= 16#0300 AND arrBuffer_FC3[9] <= 16#0308 THEN
			iStateModbus := 300;
			st_Huawei_SmartLogger[int_Poll_Counter].eErrorState := E_Huawei_SmartLogger_Error.eHuawei_SmartLoggerError;
		END_IF
	
		//Error or Timeout
		IF FPError_FC_3.Q OR timTimeout.Q THEN
			iStateModbus := 300;
			st_Huawei_SmartLogger[int_Poll_Counter].eOperatingStateInverter := E_Huawei_SmartLogger_OperatingState.Unknown;
			st_Huawei_SmartLogger[int_Poll_Counter].eErrorState	:=	E_Huawei_SmartLogger_Error.eModbusTCPError;
		END_IF
		
	12://Wait and go to step +1 or step 100
		iStateModbus_CP := iStateModbus;
		IF sint_ID_Iverter[int_Poll_Counter+1] = 0 OR int_Poll_Counter=int_maxPolls THEN		// if ID is not in use, go to state 100
			iStateModbus := 100;
		ELSE
			iStateModbus := iStateModbus+1;
			int_Poll_Counter:=int_Poll_Counter+1;			//Poll int_Poll_Counter : Inverter int_Poll_Counter 	
		END_IF
		
	13://Read out next inverter
		st_Huawei_SmartLogger[int_Poll_Counter].bFunctionIsActive := TRUE;
		iStateModbus_CP := iStateModbus;
		fbMBRead_FC3.nQuantity := 25;
		fbMBRead_FC3.nMBAddr := (51000+(25*(SINT_TO_WORD(sint_ID_Iverter[int_Poll_Counter]) - 1)));
		fbMBRead_FC3.bExecute := TRUE;
			
		IF fbMBRead_FC3.bBusy THEN 
			timDelay.IN := TRUE; 
		END_IF
		
		//Wait for Delay, copy Data and then next step
		IF NOT fbMBRead_FC3.bBusy AND NOT fbMBRead_FC3.bError AND timDelay.Q THEN
			// convert received data
			FB_ConvertData(	arrBuffer_FC3			:=	arrBuffer_FC3,
											int_Poll_Counter		:=	int_Poll_Counter,
											lrPowerTotal			=>	fbMeter[int_Poll_Counter].lrPowerTotal,	
											lrReactivePowerTotal	=> 	fbMeter[int_Poll_Counter].lrReactivePowerTotal,
											eOperatingStateInverter	=>	st_Huawei_SmartLogger[int_Poll_Counter].eOperatingStateInverter);
	
			//Next Step
			fbMBRead_FC3.bExecute := FALSE;
			timDelay.IN := FALSE;
			iStateModbus := iStateModbus+1;
			IF arrBuffer_FC3[9]<>0 THEN
				st_Huawei_SmartLogger[int_Poll_Counter].bError := FALSE; 
				st_Huawei_SmartLogger[int_Poll_Counter].eErrorState := E_Huawei_SmartLogger_Error.eNoError;
			ELSE
				st_Huawei_SmartLogger[int_Poll_Counter].bError := FALSE; 
				st_Huawei_SmartLogger[int_Poll_Counter].eErrorState := E_Huawei_SmartLogger_Error.eNoError;
			END_IF
		END_IF
			
		//Error from Inverter 1
		IF NOT fbMBRead_FC3.bBusy AND NOT fbMBRead_FC3.bError AND timDelay.Q AND arrBuffer_FC3[9] >= 16#0300 AND arrBuffer_FC3[9] <= 16#0308 THEN
			iStateModbus := 300;
			st_Huawei_SmartLogger[int_Poll_Counter].eErrorState := E_Huawei_SmartLogger_Error.eHuawei_SmartLoggerError;
		END_IF
	
		//Error or Timeout
		IF FPError_FC_3.Q OR timTimeout.Q THEN
			iStateModbus := 300;
			st_Huawei_SmartLogger[int_Poll_Counter].eOperatingStateInverter := E_Huawei_SmartLogger_OperatingState.Unknown;
			st_Huawei_SmartLogger[int_Poll_Counter].eErrorState	:=	E_Huawei_SmartLogger_Error.eModbusTCPError;
		END_IF
		
	14://Wait and go to step +1 or step 100
		iStateModbus_CP := iStateModbus;
		IF sint_ID_Iverter[int_Poll_Counter+1] = 0 OR int_Poll_Counter=int_maxPolls THEN		// if ID is not in use, go to state 100
			iStateModbus := 100;
		ELSE
			iStateModbus := iStateModbus+1;
			int_Poll_Counter:=int_Poll_Counter+1;			//Poll int_Poll_Counter : Inverter int_Poll_Counter 	
		END_IF
		
	15://Read out next inverter
		st_Huawei_SmartLogger[int_Poll_Counter].bFunctionIsActive := TRUE;
		iStateModbus_CP := iStateModbus;
		fbMBRead_FC3.nQuantity := 25;
		fbMBRead_FC3.nMBAddr := (51000+(25*(SINT_TO_WORD(sint_ID_Iverter[int_Poll_Counter]) - 1)));
		fbMBRead_FC3.bExecute := TRUE;
			
		IF fbMBRead_FC3.bBusy THEN 
			timDelay.IN := TRUE; 
		END_IF
		
		//Wait for Delay, copy Data and then next step
		IF NOT fbMBRead_FC3.bBusy AND NOT fbMBRead_FC3.bError AND timDelay.Q THEN
			// convert received data
			FB_ConvertData(	arrBuffer_FC3			:=	arrBuffer_FC3,
											int_Poll_Counter		:=	int_Poll_Counter,
											lrPowerTotal			=>	fbMeter[int_Poll_Counter].lrPowerTotal,	
											lrReactivePowerTotal	=> 	fbMeter[int_Poll_Counter].lrReactivePowerTotal,
											eOperatingStateInverter	=>	st_Huawei_SmartLogger[int_Poll_Counter].eOperatingStateInverter);
	
			//Next Step
			fbMBRead_FC3.bExecute := FALSE;
			timDelay.IN := FALSE;
			iStateModbus := iStateModbus+1;
			IF arrBuffer_FC3[9]<>0 THEN
				st_Huawei_SmartLogger[int_Poll_Counter].bError := FALSE; 
				st_Huawei_SmartLogger[int_Poll_Counter].eErrorState := E_Huawei_SmartLogger_Error.eNoError;
			ELSE
				st_Huawei_SmartLogger[int_Poll_Counter].bError := FALSE; 
				st_Huawei_SmartLogger[int_Poll_Counter].eErrorState := E_Huawei_SmartLogger_Error.eNoError;
			END_IF
		END_IF
			
		//Error from Inverter 
		IF NOT fbMBRead_FC3.bBusy AND NOT fbMBRead_FC3.bError AND timDelay.Q AND arrBuffer_FC3[9] >= 16#0300 AND arrBuffer_FC3[9] <= 16#0308 THEN
			iStateModbus := 300;
			st_Huawei_SmartLogger[int_Poll_Counter].eErrorState := E_Huawei_SmartLogger_Error.eHuawei_SmartLoggerError;
		END_IF
	
		//Error or Timeout
		IF FPError_FC_3.Q OR timTimeout.Q THEN
			iStateModbus := 300;
			st_Huawei_SmartLogger[int_Poll_Counter].eOperatingStateInverter := E_Huawei_SmartLogger_OperatingState.Unknown;
			st_Huawei_SmartLogger[int_Poll_Counter].eErrorState	:=	E_Huawei_SmartLogger_Error.eModbusTCPError;
		END_IF
		
	16://Wait and go to step +1 or step 100
		iStateModbus_CP := iStateModbus;
		IF sint_ID_Iverter[int_Poll_Counter+1] = 0 OR int_Poll_Counter=int_maxPolls THEN		// if ID is not in use, go to state 100
			iStateModbus := 100;
		ELSE
			iStateModbus := iStateModbus+1;
			int_Poll_Counter:=int_Poll_Counter+1;			//Poll int_Poll_Counter : Inverter int_Poll_Counter 	
		END_IF

	17://Read out next inverter
		st_Huawei_SmartLogger[int_Poll_Counter].bFunctionIsActive := TRUE;
		iStateModbus_CP := iStateModbus;
		fbMBRead_FC3.nQuantity := 25;
		fbMBRead_FC3.nMBAddr := (51000+(25*(SINT_TO_WORD(sint_ID_Iverter[int_Poll_Counter]) - 1)));
		fbMBRead_FC3.bExecute := TRUE;
			
		IF fbMBRead_FC3.bBusy THEN 
			timDelay.IN := TRUE; 
		END_IF
		
		//Wait for Delay, copy Data and then next step
		IF NOT fbMBRead_FC3.bBusy AND NOT fbMBRead_FC3.bError AND timDelay.Q THEN
			// convert received data
			FB_ConvertData(	arrBuffer_FC3			:=	arrBuffer_FC3,
											int_Poll_Counter		:=	int_Poll_Counter,
											lrPowerTotal			=>	fbMeter[int_Poll_Counter].lrPowerTotal,	
											lrReactivePowerTotal	=> 	fbMeter[int_Poll_Counter].lrReactivePowerTotal,
											eOperatingStateInverter	=>	st_Huawei_SmartLogger[int_Poll_Counter].eOperatingStateInverter);
	
			//Next Step
			fbMBRead_FC3.bExecute := FALSE;
			timDelay.IN := FALSE;
			iStateModbus := iStateModbus+1;
			IF arrBuffer_FC3[9]<>0 THEN
				st_Huawei_SmartLogger[int_Poll_Counter].bError := FALSE; 
				st_Huawei_SmartLogger[int_Poll_Counter].eErrorState := E_Huawei_SmartLogger_Error.eNoError;
			ELSE
				st_Huawei_SmartLogger[int_Poll_Counter].bError := FALSE; 
				st_Huawei_SmartLogger[int_Poll_Counter].eErrorState := E_Huawei_SmartLogger_Error.eNoError;
			END_IF
		END_IF
			
		//Error from Inverter 
		IF NOT fbMBRead_FC3.bBusy AND NOT fbMBRead_FC3.bError AND timDelay.Q AND arrBuffer_FC3[9] >= 16#0300 AND arrBuffer_FC3[9] <= 16#0308 THEN
			iStateModbus := 300;
			st_Huawei_SmartLogger[int_Poll_Counter].eErrorState := E_Huawei_SmartLogger_Error.eHuawei_SmartLoggerError;
		END_IF
	
		//Error or Timeout
		IF FPError_FC_3.Q OR timTimeout.Q THEN
			iStateModbus := 300;
			st_Huawei_SmartLogger[int_Poll_Counter].eOperatingStateInverter := E_Huawei_SmartLogger_OperatingState.Unknown;
			st_Huawei_SmartLogger[int_Poll_Counter].eErrorState	:=	E_Huawei_SmartLogger_Error.eModbusTCPError;
		END_IF
		
	18://Wait and go to step +1 or step 100
		iStateModbus_CP := iStateModbus;
		IF sint_ID_Iverter[int_Poll_Counter+1] = 0 OR int_Poll_Counter=int_maxPolls THEN		// if ID is not in use, go to state 100
			iStateModbus := 100;
		ELSE
			iStateModbus := iStateModbus+1;
			int_Poll_Counter:=int_Poll_Counter+1;			//Poll int_Poll_Counter : Inverter int_Poll_Counter 	
		END_IF
		
	19://Read out next inverter
		st_Huawei_SmartLogger[int_Poll_Counter].bFunctionIsActive := TRUE;
		iStateModbus_CP := iStateModbus;
		fbMBRead_FC3.nQuantity := 25;
		fbMBRead_FC3.nMBAddr := (51000+(25*(SINT_TO_WORD(sint_ID_Iverter[int_Poll_Counter]) - 1)));
		fbMBRead_FC3.bExecute := TRUE;
			
		IF fbMBRead_FC3.bBusy THEN 
			timDelay.IN := TRUE; 
		END_IF
		
		//Wait for Delay, copy Data and then next step
		IF NOT fbMBRead_FC3.bBusy AND NOT fbMBRead_FC3.bError AND timDelay.Q THEN
			// convert received data
			FB_ConvertData(	arrBuffer_FC3			:=	arrBuffer_FC3,
											int_Poll_Counter		:=	int_Poll_Counter,
											lrPowerTotal			=>	fbMeter[int_Poll_Counter].lrPowerTotal,	
											lrReactivePowerTotal	=> 	fbMeter[int_Poll_Counter].lrReactivePowerTotal,
											eOperatingStateInverter	=>	st_Huawei_SmartLogger[int_Poll_Counter].eOperatingStateInverter);
	
			//Next Step
			fbMBRead_FC3.bExecute := FALSE;
			timDelay.IN := FALSE;
			iStateModbus := iStateModbus+1;
			IF arrBuffer_FC3[9]<>0 THEN
				st_Huawei_SmartLogger[int_Poll_Counter].bError := FALSE; 
				st_Huawei_SmartLogger[int_Poll_Counter].eErrorState := E_Huawei_SmartLogger_Error.eNoError;
			ELSE
				st_Huawei_SmartLogger[int_Poll_Counter].bError := FALSE; 
				st_Huawei_SmartLogger[int_Poll_Counter].eErrorState := E_Huawei_SmartLogger_Error.eNoError;
			END_IF
		END_IF
			
		//Error or Timeout
		IF FPError_FC_3.Q OR timTimeout.Q THEN
			iStateModbus := 300;
			st_Huawei_SmartLogger[int_Poll_Counter].eOperatingStateInverter := E_Huawei_SmartLogger_OperatingState.Unknown;
			st_Huawei_SmartLogger[int_Poll_Counter].eErrorState	:=	E_Huawei_SmartLogger_Error.eModbusTCPError;
		END_IF
	
		//Error or Timeout
		IF FPError_FC_3.Q OR timTimeout.Q THEN
			iStateModbus := 300;
			st_Huawei_SmartLogger[int_Poll_Counter].eOperatingStateInverter := E_Huawei_SmartLogger_Error.eModbusTCPError;
		END_IF

	20://Wait and go to step +1 or step 100
		iStateModbus_CP := iStateModbus;
		IF sint_ID_Iverter[int_Poll_Counter+1] = 0 OR int_Poll_Counter=int_maxPolls THEN		// if ID is not in use, go to state 100
			iStateModbus := 100;
		ELSE
			iStateModbus := iStateModbus+1;
			int_Poll_Counter:=int_Poll_Counter+1;			//Poll int_Poll_Counter : Inverter int_Poll_Counter 	
		END_IF

	21://Read out next inverter
		st_Huawei_SmartLogger[int_Poll_Counter].bFunctionIsActive := TRUE;
		iStateModbus_CP := iStateModbus;
		fbMBRead_FC3.nQuantity := 25;
		fbMBRead_FC3.nMBAddr := (51000+(25*(SINT_TO_WORD(sint_ID_Iverter[int_Poll_Counter]) - 1)));
		fbMBRead_FC3.bExecute := TRUE;
			
		IF fbMBRead_FC3.bBusy THEN 
			timDelay.IN := TRUE; 
		END_IF
		
		//Wait for Delay, copy Data and then next step
		IF NOT fbMBRead_FC3.bBusy AND NOT fbMBRead_FC3.bError AND timDelay.Q THEN
			// convert received data
			FB_ConvertData(	arrBuffer_FC3			:=	arrBuffer_FC3,
											int_Poll_Counter		:=	int_Poll_Counter,
											lrPowerTotal			=>	fbMeter[int_Poll_Counter].lrPowerTotal,	
											lrReactivePowerTotal	=> 	fbMeter[int_Poll_Counter].lrReactivePowerTotal,
											eOperatingStateInverter	=>	st_Huawei_SmartLogger[int_Poll_Counter].eOperatingStateInverter);
	
			//Next Step
			fbMBRead_FC3.bExecute := FALSE;
			timDelay.IN := FALSE;
			iStateModbus := iStateModbus+1;
			IF arrBuffer_FC3[9]<>0 THEN
				st_Huawei_SmartLogger[int_Poll_Counter].bError := FALSE; 
				st_Huawei_SmartLogger[int_Poll_Counter].eErrorState := E_Huawei_SmartLogger_Error.eNoError;
			ELSE
				st_Huawei_SmartLogger[int_Poll_Counter].bError := FALSE; 
				st_Huawei_SmartLogger[int_Poll_Counter].eErrorState := E_Huawei_SmartLogger_Error.eNoError;
			END_IF
		END_IF
			
		//Error from Inverter 
		IF NOT fbMBRead_FC3.bBusy AND NOT fbMBRead_FC3.bError AND timDelay.Q AND arrBuffer_FC3[9] >= 16#0300 AND arrBuffer_FC3[9] <= 16#0308 THEN
			iStateModbus := 300;
			st_Huawei_SmartLogger[int_Poll_Counter].eErrorState := E_Huawei_SmartLogger_Error.eHuawei_SmartLoggerError;
		END_IF
	
		//Error or Timeout
		IF FPError_FC_3.Q OR timTimeout.Q THEN
			iStateModbus := 300;
			st_Huawei_SmartLogger[int_Poll_Counter].eOperatingStateInverter := E_Huawei_SmartLogger_OperatingState.Unknown;
			st_Huawei_SmartLogger[int_Poll_Counter].eErrorState	:=	E_Huawei_SmartLogger_Error.eModbusTCPError;
		END_IF
		
	22://Wait and go to step +1 or step 100
		iStateModbus_CP := iStateModbus;
		IF sint_ID_Iverter[int_Poll_Counter+1] = 0 OR int_Poll_Counter=int_maxPolls THEN		// if ID is not in use, go to state 100
			iStateModbus := 100;
		ELSE
			iStateModbus := iStateModbus+1;
			int_Poll_Counter:=int_Poll_Counter+1;			//Poll int_Poll_Counter : Inverter int_Poll_Counter 	
		END_IF

	23://Read out next inverter
		st_Huawei_SmartLogger[int_Poll_Counter].bFunctionIsActive := TRUE;
		iStateModbus_CP := iStateModbus;
		fbMBRead_FC3.nQuantity := 25;
		fbMBRead_FC3.nMBAddr := (51000+(25*(SINT_TO_WORD(sint_ID_Iverter[int_Poll_Counter]) - 1)));
		fbMBRead_FC3.bExecute := TRUE;
			
		IF fbMBRead_FC3.bBusy THEN 
			timDelay.IN := TRUE; 
		END_IF
		
		//Wait for Delay, copy Data and then next step
		IF NOT fbMBRead_FC3.bBusy AND NOT fbMBRead_FC3.bError AND timDelay.Q THEN
			// convert received data
			FB_ConvertData(	arrBuffer_FC3			:=	arrBuffer_FC3,
											int_Poll_Counter		:=	int_Poll_Counter,
											lrPowerTotal			=>	fbMeter[int_Poll_Counter].lrPowerTotal,	
											lrReactivePowerTotal	=> 	fbMeter[int_Poll_Counter].lrReactivePowerTotal,
											eOperatingStateInverter	=>	st_Huawei_SmartLogger[int_Poll_Counter].eOperatingStateInverter);
	
			//Next Step
			fbMBRead_FC3.bExecute := FALSE;
			timDelay.IN := FALSE;
			iStateModbus := iStateModbus+1;
			IF arrBuffer_FC3[9]<>0 THEN
				st_Huawei_SmartLogger[int_Poll_Counter].bError := FALSE; 
				st_Huawei_SmartLogger[int_Poll_Counter].eErrorState := E_Huawei_SmartLogger_Error.eNoError;
			ELSE
				st_Huawei_SmartLogger[int_Poll_Counter].bError := FALSE; 
				st_Huawei_SmartLogger[int_Poll_Counter].eErrorState := E_Huawei_SmartLogger_Error.eNoError;
			END_IF
		END_IF
			
		//Error from Inverter 
		IF NOT fbMBRead_FC3.bBusy AND NOT fbMBRead_FC3.bError AND timDelay.Q AND arrBuffer_FC3[9] >= 16#0300 AND arrBuffer_FC3[9] <= 16#0308 THEN
			iStateModbus := 300;
			st_Huawei_SmartLogger[int_Poll_Counter].eErrorState := E_Huawei_SmartLogger_Error.eHuawei_SmartLoggerError;
		END_IF
	
		//Error or Timeout
		IF FPError_FC_3.Q OR timTimeout.Q THEN
			iStateModbus := 300;
			st_Huawei_SmartLogger[int_Poll_Counter].eOperatingStateInverter := E_Huawei_SmartLogger_OperatingState.Unknown;
			st_Huawei_SmartLogger[int_Poll_Counter].eErrorState	:=	E_Huawei_SmartLogger_Error.eModbusTCPError;
		END_IF
		
	24://Wait and go to step +1 or step 100
		iStateModbus_CP := iStateModbus;
		IF sint_ID_Iverter[int_Poll_Counter+1] = 0 OR int_Poll_Counter=int_maxPolls THEN		// if ID is not in use, go to state 100
			iStateModbus := 100;
		ELSE
			iStateModbus := iStateModbus+1;
			int_Poll_Counter:=int_Poll_Counter+1;			//Poll int_Poll_Counter : Inverter int_Poll_Counter 	
		END_IF




		
		
		
	100://Wait and go to step 1 
		iStateModbus_CP := iStateModbus;
		ton_Wait.In:=TRUE;
		IF ton_Wait.Q THEN
			ton_Wait.In:=FALSE;
			iStateModbus := 1;
		END_IF
			
	300://Error
		iStateModbus_CP := iStateModbus;
		timDelay.IN := FALSE;
		fbMBRead_FC3.bExecute := FALSE;
		st_Huawei_SmartLogger[int_Poll_Counter].bError := TRUE;
		ton_Wait.In:=TRUE;
		IF ton_Wait.Q THEN
			ton_Wait.In:=FALSE;
			iStateModbus := 1;
		END_IF
END_CASE

// wait timer
ton_Wait(PT:=T#2S);

	

(*------------------------------------------------------------------------------------------Modbus TCP Function---------------------------------------------------------------------------------------------*)

fbMBRead_FC3(	sIPAddr:= sIPAdress, 
				nTCPPort:= 502, 
				nUnitID := 0,
				cbLength:= SIZEOF(arrBuffer_FC3), 
				pDestAddr:= ADR(arrBuffer_FC3), 
				tTimeout:= T#10S );

FPError_FC_3(CLK:= fbMBRead_FC3.bError, Q=> );

(*----------------------------------------------------------------------------------------Electric Meter Data----------------------------------------------------------------------------------------------*)

//Error and Warning
FOR x:=1 TO 20 BY 1 DO
	IF timDissableFunctions.Q THEN 
		fbMeter[x].bWarning := TRUE; 
		fbMeter[x].iWarningCode := 0; 
	ELSE 
		fbMeter[x].bWarning := FALSE; 
	END_IF   

	IF st_Huawei_SmartLogger[x].bError OR Lynus_Standards.GVL_Energy.stNumberOfDevices.diNumberOfElectricMeters > Constants_Energy.diMaxNumberOfElectricMeters THEN 
		fbMeter[x].bError := TRUE; 
	ELSE 
		fbMeter[x].bError := FALSE; 
	END_IF  

	IF Lynus_Standards.GVL_Energy.stNumberOfDevices.diNumberOfElectricMeters > Constants_Energy.diMaxNumberOfElectricMeters THEN 
		fbMeter[x].iErrorCode := 1;
	ELSIF st_Huawei_SmartLogger[x].bError THEN 
		fbMeter[x].iErrorCode := 0;
	END_IF  

	//Function block for meter data
	fbMeter[x](
		bEnable:= bEnable AND NOT timDissableFunctions.Q, 
		bError:= , 
		bEnableReadOutFunction:= TRUE, 
		bWriteWithDelay:= TRUE,
		bPowerDataInvers:= TRUE, 
		bReadOutDataDone:= TRUE,
		iTimeReadOutInterval:= , 
		iErrorCode:= , 
		iWarningCode:= , 
		lrTotalCounterEnergy_Consumption:= 0, 
		lrTotalCounterEnergy_Production:= , 
		lrCounterEnergyT1_Consumption:= 0, 
		lrCounterEnergyT2_Consumption:= 0, 
		lrCounterEnergyT1_Production:= , 
		lrCounterEnergyT2_Production:= 0, 
		lrCurrentL1:= , 
		lrVoltageL1N:= , 
		lrVoltageL1L2:= , 
		lrPowerL1:= 0, 
		lrCurrentL2:= , 
		lrVoltageL2N:= , 
		lrVoltageL2L3:= , 
		lrPowerL2:= 0, 
		lrCurrentL3:= , 
		lrVoltageL3N:= , 
		lrVoltageL3L1:= , 
		lrPowerL3:= 0, 
		lrPowerTotal:= , 
		lrFrequency:= , 
		lrReactivePowerTotal:= , 
		lrApparentPowerTotal:= , 
		tTimDelayOutput:= T#5S, 
		stDataEMOutPower=> , 
		stDataEMOutPowerDelay=> stDataEMPower_PV[x], 
		stDataEMOutCounter=> ,
		stDataEMOutCounterDelay=> stDataEMCounter_PV[x], 
		bReadOutMeter=> );

END_FOR
//Read Out Data done for EM Function
IF NOT fbMBRead_FC3.bBusy AND NOT fbMBRead_FC3.bError THEN 
	fbMeter[int_Poll_Counter].bReadOutDataDone := TRUE;
ELSE 
	fbMeter[int_Poll_Counter].bReadOutDataDone := FALSE;
END_IF



(*-----------------------------------------------------------Handle data to Global structure for the Electric Meter system-----------------------------------------------------------------*)

CASE iStateGVLData OF
	
	0://Init Step
		byWaitInStep := 0;
		diCounterForGVL := 1;
	
	1://Wait for 4 Steps before clean al Data on GVL
		byWaitInStep := byWaitInStep + 1;
		IF byWaitInStep >= 4 AND fbNumberDevice.bNumberIsCalculatet THEN 
			iStateGVLData := 2; 
		END_IF
		//To much Devices, back to the Init step
		IF byWaitInStep >= 4 AND NOT fbNumberDevice.bNumberIsCalculatet THEN 
			iStateGVLData := 0; 
		END_IF	
			
	2://Clear all Data in GVL
		Lynus_Standards.GVL_Energy.stDataElectricMeters[diCounterForGVL].bEnabled := FALSE;	
		Lynus_Standards.GVL_Energy.stDataElectricMeters[diCounterForGVL].byErrorWarning := 0;
		Lynus_Standards.GVL_Energy.stDataElectricMeters[diCounterForGVL].lrCounterEnergyT1_Consumption := 0;
		Lynus_Standards.GVL_Energy.stDataElectricMeters[diCounterForGVL].lrCounterEnergyT1_Production := 0;
		Lynus_Standards.GVL_Energy.stDataElectricMeters[diCounterForGVL].lrCounterEnergyT2_Consumption := 0;
		Lynus_Standards.GVL_Energy.stDataElectricMeters[diCounterForGVL].lrCounterEnergyT2_Production := 0;
		Lynus_Standards.GVL_Energy.stDataElectricMeters[diCounterForGVL].lrPower := 0;
		Lynus_Standards.GVL_Energy.stDataElectricMeters[diCounterForGVL].lrPowerConsumption := 0;
		Lynus_Standards.GVL_Energy.stDataElectricMeters[diCounterForGVL].lrPowerConsumption := 0;
		Lynus_Standards.GVL_Energy.stDataElectricMeters[diCounterForGVL].lrPowerProduction := 0;
		Lynus_Standards.GVL_Energy.stDataElectricMeters[diCounterForGVL].lrTotalCounterEnergy_Consumption := 0;
		Lynus_Standards.GVL_Energy.stDataElectricMeters[diCounterForGVL].lrTotalCounterEnergy_Production := 0;
		
		diCounterForGVL := diCounterForGVL + 1;
		diCounterForGVL := LIMIT(0,diCounterForGVL,Constants_Energy.diMaxNumberOfElectricMeters);
		//Back to the init step
		IF diCounterForGVL >= Constants_Energy.diMaxNumberOfElectricMeters THEN 
			iStateGVLData := 0; 
		END_IF
END_CASE 	 

IF diNrOfEM_OUT_PV > 0 AND fbNumberDevice.bNumberIsCalculatet THEN
	Lynus_Standards.GVL_Energy.stDataElectricMeters[diNrOfEM_OUT_PV].bEnabled := fbElMeter.stDataEMOutPower.bEnabled;
	Lynus_Standards.GVL_Energy.stDataElectricMeters[diNrOfEM_OUT_PV].byErrorWarning := fbElMeter.stDataEMOutPower.byErrorWarning;
	Lynus_Standards.GVL_Energy.stDataElectricMeters[diNrOfEM_OUT_PV].lrCounterEnergyT1_Consumption := fbElMeter.stDataEMOutCounter.lrCounterEnergyT1_Consumption;
	Lynus_Standards.GVL_Energy.stDataElectricMeters[diNrOfEM_OUT_PV].lrCounterEnergyT1_Production := fbElMeter.stDataEMOutCounter.lrCounterEnergyT1_Production;
	Lynus_Standards.GVL_Energy.stDataElectricMeters[diNrOfEM_OUT_PV].lrCounterEnergyT2_Consumption := fbElMeter.stDataEMOutCounter.lrCounterEnergyT2_Consumption;
	Lynus_Standards.GVL_Energy.stDataElectricMeters[diNrOfEM_OUT_PV].lrCounterEnergyT2_Production := fbElMeter.stDataEMOutCounter.lrCounterEnergyT2_Production;		
	Lynus_Standards.GVL_Energy.stDataElectricMeters[diNrOfEM_OUT_PV].lrPower := fbElMeter.lrPowerTotal; // fbElMeter.stDataEMOutPower.lrPowerTotal;
	Lynus_Standards.GVL_Energy.stDataElectricMeters[diNrOfEM_OUT_PV].lrPowerConsumption := fbElMeter.stDataEMOutPower.lrPowerConsumption;
	Lynus_Standards.GVL_Energy.stDataElectricMeters[diNrOfEM_OUT_PV].lrPowerProduction := fbElMeter.stDataEMOutPower.lrPowerProduction;
	Lynus_Standards.GVL_Energy.stDataElectricMeters[diNrOfEM_OUT_PV].lrTotalCounterEnergy_Consumption := fbElMeter.stDataEMOutCounter.lrTotalCounterEnergy_Consumption;
	Lynus_Standards.GVL_Energy.stDataElectricMeters[diNrOfEM_OUT_PV].lrTotalCounterEnergy_Production := fbElMeter.stDataEMOutCounter.lrTotalCounterEnergy_Production;
END_IF


// Sum values for Meter
fbElMeter.lrPowerTotal := 0;
FOR byLPForInverter := 1 TO 20 BY 1 DO 
	lrCounterEnergyProduction := lrCounterEnergyProduction + fbMeter[byLPForInverter].stDataEMOutCounterDelay.lrTotalCounterEnergy_Production;
	IF lrCounterEnergyProduction > fbElMeter.lrCounterEnergyT1_Production THEN
		fbElMeter.lrCounterEnergyT1_Production := lrCounterEnergyProduction;
	END_IF
	fbElMeter.lrPowerTotal := fbElMeter.lrPowerTotal + fbMeter[byLPForInverter].stDataEMOutPowerDelay.lrPowerTotal;
END_FOR	
					
fbElMeter.lrTotalCounterEnergy_Production := fbElMeter.lrCounterEnergyT1_Production; 
fbElMeter(bEnable:=TRUE);


